LIN {X 0,Y 560.039,Z 923.26,A -85,B 0,C 180,E1 27100.284,E2 27100.284} C_VEL
LIN {X 0,Y 559.963,Z 930.88,A -85,B 0,C 180,E1 27098.213,E2 27098.213} C_VEL
LIN {X 0,Y 559.931,Z 936.64,A -85,B 0,C 180,E1 27096.151,E2 27096.151} C_VEL
LIN {X 0,Y 559.918,Z 940.7,A -85,B 0,C 180,E1 27094.096,E2 27094.096} C_VEL
LIN {X 0,Y 559.916,Z 943.21,A -85,B 0,C 180,E1 27091.944,E2 27091.944} C_VEL
LIN {X 0,Y 559.914,Z 943.994,A -85,B 0,C 180,E1 27089.898,E2 27089.898} C_VEL
LIN {X 0,Y 559.91,Z 943.066,A -85,B 0,C 180,E1 27087.748,E2 27087.748} C_VEL
LIN {X 0,Y 559.917,Z 940.522,A -85,B 0,C 180,E1 27085.699,E2 27085.699} C_VEL
LIN {X 0,Y 559.934,Z 936.354,A -85,B 0,C 180,E1 27083.644,E2 27083.644} C_VEL
LIN {X 0,Y 559.973,Z 930.444,A -85,B 0,C 180,E1 27081.57,E2 27081.57} C_VEL
LIN {X 0,Y 560.039,Z 923.202,A -85,B 0,C 180,E1 27079.612,E2 27079.612} C_VEL
LIN {X 0,Y 560.173,Z 913.998,A -85,B 0,C 180,E1 27077.632,E2 27077.632} C_VEL
LIN {X 0,Y 560.353,Z 903.373,A -85,B 0,C 180,E1 27075.745,E2 27075.745} C_VEL
LIN {X 0,Y 560.607,Z 891.369,A -85,B 0,C 180,E1 27073.952,E2 27073.952} C_VEL
LIN {X 0,Y 560.935,Z 877.981,A -85,B 0,C 180,E1 27072.253,E2 27072.253} C_VEL
LIN {X 0,Y 561.332,Z 863.174,A -85,B 0,C 180,E1 27070.652,E2 27070.652} C_VEL
LIN {X 0,Y 561.802,Z 846.535,A -85,B 0,C 180,E1 27069.126,E2 27069.126} C_VEL
LIN {X 0,Y 562.324,Z 828.625,A -85,B 0,C 180,E1 27067.745,E2 27067.745} C_VEL
LIN {X 0,Y 562.836,Z 809.963,A -85,B 0,C 180,E1 27066.551,E2 27066.551} C_VEL
LIN {X 0,Y 563.315,Z 791.261,A -85,B 0,C 180,E1 27065.571,E2 27065.571} C_VEL
LIN {X 0,Y 563.724,Z 772.173,A -85,B 0,C 180,E1 27064.766,E2 27064.766} C_VEL
LIN {X 0,Y 564.117,Z 751.599,A -85,B 0,C 180,E1 27064.104,E2 27064.104} C_VEL
LIN {X 0,Y 564.417,Z 731.328,A -85,B 0,C 180,E1 27063.645,E2 27063.645} C_VEL
LIN {X 0,Y 565.685,Z 480.008,A -85,B 0,C 180,E1 27060.141,E2 27060.141} C_VEL
LIN {X 0,Y 565.144,Z 474.616,A -85,B 0,C 180,E1 27060.032,E2 27060.032} C_VEL
LIN {X 0,Y 564.411,Z 469.546,A -85,B 0,C 180,E1 27059.882,E2 27059.882} C_VEL
LIN {X 0,Y 565.386,Z 421.661,A -85,B 0,C 180,E1 27056.633,E2 27056.633} C_VEL
LIN {X 0,Y 566.258,Z 392.209,A -85,B 0,C 180,E1 27054.54,E2 27054.54} C_VEL
LIN {X 0,Y 562.618,Z 383.241,A -85,B 0,C 180,E1 27053.53,E2 27053.53} C_VEL
LIN {X 0,Y 560.275,Z 377.562,A -85,B 0,C 180,E1 27052.843,E2 27052.843} C_VEL
LIN {X 0,Y 560.267,Z 377.245,A -85,B 0,C 180,E1 27051.868,E2 27051.868} C_VEL
LIN {X 0,Y 560.221,Z 377.251,A -85,B 0,C 180,E1 27048.808,E2 27048.808} C_VEL
LIN {X 0,Y 560.261,Z 377.247,A -85,B 0,C 180,E1 27045.549,E2 27045.549} C_VEL
LIN {X 0,Y 560.226,Z 377.259,A -85,B 0,C 180,E1 27042.426,E2 27042.426} C_VEL
LIN {X 0,Y 560.237,Z 377.262,A -85,B 0,C 180,E1 27039.051,E2 27039.051} C_VEL
LIN {X 0,Y 560.23,Z 377.247,A -85,B 0,C 180,E1 27036.051,E2 27036.051} C_VEL
LIN {X 0,Y 560.224,Z 377.259,A -85,B 0,C 180,E1 27032.605,E2 27032.605} C_VEL
LIN {X 0,Y 560.252,Z 377.242,A -85,B 0,C 180,E1 27029.51,E2 27029.51} C_VEL
LIN {X 0,Y 560.218,Z 377.258,A -85,B 0,C 180,E1 27026.272,E2 27026.272} C_VEL
LIN {X 0,Y 560.268,Z 377.258,A -85,B 0,C 180,E1 27023.118,E2 27023.118} C_VEL
LIN {X 0,Y 560.214,Z 377.26,A -85,B 0,C 180,E1 27019.932,E2 27019.932} C_VEL
LIN {X 0,Y 560.273,Z 377.257,A -85,B 0,C 180,E1 27016.805,E2 27016.805} C_VEL
LIN {X 0,Y 560.211,Z 377.26,A -85,B 0,C 180,E1 27013.627,E2 27013.627} C_VEL
LIN {X 0,Y 560.274,Z 377.254,A -85,B 0,C 180,E1 27010.48,E2 27010.48} C_VEL
LIN {X 0,Y 560.208,Z 377.257,A -85,B 0,C 180,E1 27007.28,E2 27007.28} C_VEL
LIN {X 0,Y 560.28,Z 377.258,A -85,B 0,C 180,E1 27004.094,E2 27004.094} C_VEL
LIN {X 0,Y 560.207,Z 377.259,A -85,B 0,C 180,E1 27000.921,E2 27000.921} C_VEL
LIN {X 0,Y 560.278,Z 377.261,A -85,B 0,C 180,E1 26997.75,E2 26997.75} C_VEL
LIN {X 0,Y 560.205,Z 377.26,A -85,B 0,C 180,E1 26994.572,E2 26994.572} C_VEL
LIN {X 0,Y 560.269,Z 377.26,A -85,B 0,C 180,E1 26991.37,E2 26991.37} C_VEL
LIN {X 0,Y 560.204,Z 377.253,A -85,B 0,C 180,E1 26988.261,E2 26988.261} C_VEL
LIN {X 0,Y 560.254,Z 377.258,A -85,B 0,C 180,E1 26985.003,E2 26985.003} C_VEL
LIN {X 0,Y 560.203,Z 377.256,A -85,B 0,C 180,E1 26982.015,E2 26982.015} C_VEL
LIN {X 0,Y 560.256,Z 377.257,A -85,B 0,C 180,E1 26978.76,E2 26978.76} C_VEL
LIN {X 0,Y 560.201,Z 377.256,A -85,B 0,C 180,E1 26975.764,E2 26975.764} C_VEL
LIN {X 0,Y 560.255,Z 377.262,A -85,B 0,C 180,E1 26972.496,E2 26972.496} C_VEL
LIN {X 0,Y 560.2,Z 377.25,A -85,B 0,C 180,E1 26969.425,E2 26969.425} C_VEL
LIN {X 0,Y 560.245,Z 377.256,A -85,B 0,C 180,E1 26966.164,E2 26966.164} C_VEL
LIN {X 0,Y 560.202,Z 377.263,A -85,B 0,C 180,E1 26963.092,E2 26963.092} C_VEL
LIN {X 0,Y 560.233,Z 377.255,A -85,B 0,C 180,E1 26959.806,E2 26959.806} C_VEL
LIN {X 0,Y 560.196,Z 377.245,A -85,B 0,C 180,E1 26956.876,E2 26956.876} C_VEL
LIN {X 0,Y 560.287,Z 377.452,A -85,B 0,C 180,E1 26956.18,E2 26956.18} C_VEL
LIN {X 0,Y 561.118,Z 379.974,A -85,B 0,C 180,E1 26955.899,E2 26955.899} C_VEL
LIN {X 0,Y 564.918,Z 386.463,A -85,B 0,C 180,E1 26955.214,E2 26955.214} C_VEL
LIN {X 0,Y 570.593,Z 397.019,A -85,B 0,C 180,E1 26954.056,E2 26954.056} C_VEL
LIN {X 0,Y 569.301,Z 451.788,A -85,B 0,C 180,E1 26951.15,E2 26951.15} C_VEL
LIN {X 0,Y 569.17,Z 466.355,A -85,B 0,C 180,E1 26950.418,E2 26950.418} C_VEL
LIN {X 0,Y 570.273,Z 475.671,A -85,B 0,C 180,E1 26950.173,E2 26950.173} C_VEL
LIN {X 0,Y 568.787,Z 680.489,A -85,B 0,C 180,E1 26947.054,E2 26947.054} C_VEL
LIN {X 0,Y 567.809,Z 815.971,A -85,B 0,C 180,E1 26945.018,E2 26945.018} C_VEL
LIN {X 0,Y 567.322,Z 839.745,A -85,B 0,C 180,E1 26944.473,E2 26944.473} C_VEL
LIN {X 0,Y 566.852,Z 861.613,A -85,B 0,C 180,E1 26943.785,E2 26943.785} C_VEL
LIN {X 0,Y 566.166,Z 883.682,A -85,B 0,C 180,E1 26942.892,E2 26942.892} C_VEL
LIN {X 0,Y 565.506,Z 904.783,A -85,B 0,C 180,E1 26941.855,E2 26941.855} C_VEL
LIN {X 0,Y 564.723,Z 925.843,A -85,B 0,C 180,E1 26940.605,E2 26940.605} C_VEL
LIN {X 0,Y 563.96,Z 946.403,A -85,B 0,C 180,E1 26939.18,E2 26939.18} C_VEL
LIN {X 0,Y 563.25,Z 964.586,A -85,B 0,C 180,E1 26937.716,E2 26937.716} C_VEL
LIN {X 0,Y 562.525,Z 983.959,A -85,B 0,C 180,E1 26935.923,E2 26935.923} C_VEL
LIN {X 0,Y 561.904,Z 1001.171,A -85,B 0,C 180,E1 26934.101,E2 26934.101} C_VEL
LIN {X 0,Y 561.359,Z 1017.098,A -85,B 0,C 180,E1 26932.152,E2 26932.152} C_VEL
LIN {X 0,Y 560.903,Z 1032.335,A -85,B 0,C 180,E1 26930.015,E2 26930.015} C_VEL
LIN {X 0,Y 560.562,Z 1045.006,A -85,B 0,C 180,E1 26927.974,E2 26927.974} C_VEL
LIN {X 0,Y 560.296,Z 1056.318,A -85,B 0,C 180,E1 26925.845,E2 26925.845} C_VEL
LIN {X 0,Y 560.126,Z 1065.995,A -85,B 0,C 180,E1 26923.734,E2 26923.734} C_VEL
LIN {X 0,Y 560.023,Z 1074.34,A -85,B 0,C 180,E1 26921.535,E2 26921.535} C_VEL
LIN {X 0,Y 559.945,Z 1080.869,A -85,B 0,C 180,E1 26919.455,E2 26919.455} C_VEL
LIN {X 0,Y 559.899,Z 1086.634,A -85,B 0,C 180,E1 26917.078,E2 26917.078} C_VEL
LIN {X 0,Y 559.911,Z 1090.276,A -85,B 0,C 180,E1 26915.02,E2 26915.02} C_VEL
LIN {X 0,Y 559.913,Z 1092.988,A -85,B 0,C 180,E1 26912.559,E2 26912.559} C_VEL
LIN {X 0,Y 559.887,Z 1093.917,A -85,B 0,C 180,E1 26910.409,E2 26910.409} C_VEL
LIN {X 0,Y 559.912,Z 1093.324,A -85,B 0,C 180,E1 26907.953,E2 26907.953} C_VEL
LIN {X 0,Y 559.912,Z 1091.276,A -85,B 0,C 180,E1 26905.699,E2 26905.699} C_VEL
LIN {X 0,Y 559.914,Z 1087.46,A -85,B 0,C 180,E1 26903.334,E2 26903.334} C_VEL
LIN {X 0,Y 559.949,Z 1082.806,A -85,B 0,C 180,E1 26901.27,E2 26901.27} C_VEL
LIN {X 0,Y 559.994,Z 1075.764,A -85,B 0,C 180,E1 26898.882,E2 26898.882} C_VEL
LIN {X 0,Y 560.096,Z 1068.109,A -85,B 0,C 180,E1 26896.791,E2 26896.791} C_VEL
LIN {X 0,Y 560.276,Z 1057.882,A -85,B 0,C 180,E1 26894.473,E2 26894.473} C_VEL
LIN {X 0,Y 560.533,Z 1046.819,A -85,B 0,C 180,E1 26892.348,E2 26892.348} C_VEL
LIN {X 0,Y 560.861,Z 1033.752,A -85,B 0,C 180,E1 26890.201,E2 26890.201} C_VEL
LIN {X 0,Y 561.294,Z 1019.336,A -85,B 0,C 180,E1 26888.136,E2 26888.136} C_VEL
LIN {X 0,Y 561.8,Z 1003.941,A -85,B 0,C 180,E1 26886.227,E2 26886.227} C_VEL
LIN {X 0,Y 562.437,Z 986.114,A -85,B 0,C 180,E1 26884.293,E2 26884.293} C_VEL
LIN {X 0,Y 563.119,Z 968.256,A -85,B 0,C 180,E1 26882.595,E2 26882.595} C_VEL
LIN {X 0,Y 563.847,Z 949.336,A -85,B 0,C 180,E1 26881.046,E2 26881.046} C_VEL
LIN {X 0,Y 564.609,Z 928.601,A -85,B 0,C 180,E1 26879.57,E2 26879.57} C_VEL
LIN {X 0,Y 565.354,Z 908.827,A -85,B 0,C 180,E1 26878.373,E2 26878.373} C_VEL
LIN {X 0,Y 566.073,Z 886.169,A -85,B 0,C 180,E1 26877.22,E2 26877.22} C_VEL
LIN {X 0,Y 566.734,Z 865.501,A -85,B 0,C 180,E1 26876.36,E2 26876.36} C_VEL
LIN {X 0,Y 567.276,Z 842.338,A -85,B 0,C 180,E1 26875.6,E2 26875.6} C_VEL
LIN {X 0,Y 567.747,Z 820.122,A -85,B 0,C 180,E1 26875.058,E2 26875.058} C_VEL
LIN {X 0,Y 568.087,Z 782.758,A -85,B 0,C 180,E1 26874.465,E2 26874.465} C_VEL
LIN {X 0,Y 569.521,Z 575.861,A -85,B 0,C 180,E1 26871.366,E2 26871.366} C_VEL
LIN {X 0,Y 570.109,Z 472.892,A -85,B 0,C 180,E1 26869.768,E2 26869.768} C_VEL
LIN {X 0,Y 569.041,Z 464.13,A -85,B 0,C 180,E1 26869.491,E2 26869.491} C_VEL
LIN {X 0,Y 570.379,Z 406.466,A -85,B 0,C 180,E1 26866.455,E2 26866.455} C_VEL
LIN {X 0,Y 570.536,Z 396.902,A -85,B 0,C 180,E1 26865.932,E2 26865.932} C_VEL
LIN {X 0,Y 564.905,Z 386.448,A -85,B 0,C 180,E1 26864.784,E2 26864.784} C_VEL
LIN {X 0,Y 562.383,Z 381.983,A -85,B 0,C 180,E1 26864.323,E2 26864.323} C_VEL
LIN {X 0,Y 560.392,Z 377.966,A -85,B 0,C 180,E1 26863.909,E2 26863.909} C_VEL
LIN {X 0,Y 560.241,Z 377.261,A -85,B 0,C 180,E1 26863.683,E2 26863.683} C_VEL
LIN {X 0,Y 560.2,Z 377.267,A -85,B 0,C 180,E1 26860.651,E2 26860.651} C_VEL
LIN {X 0,Y 560.236,Z 377.263,A -85,B 0,C 180,E1 26857.358,E2 26857.358} C_VEL
LIN {X 0,Y 560.201,Z 377.256,A -85,B 0,C 180,E1 26854.333,E2 26854.333} C_VEL
LIN {X 0,Y 560.231,Z 377.248,A -85,B 0,C 180,E1 26851.049,E2 26851.049} C_VEL
LIN {X 0,Y 560.203,Z 377.263,A -85,B 0,C 180,E1 26848.111,E2 26848.111} C_VEL
LIN {X 0,Y 560.236,Z 377.255,A -85,B 0,C 180,E1 26844.797,E2 26844.797} C_VEL
LIN {X 0,Y 560.202,Z 377.262,A -85,B 0,C 180,E1 26841.857,E2 26841.857} C_VEL
LIN {X 0,Y 560.248,Z 377.254,A -85,B 0,C 180,E1 26838.618,E2 26838.618} C_VEL
LIN {X 0,Y 560.202,Z 377.261,A -85,B 0,C 180,E1 26835.635,E2 26835.635} C_VEL
LIN {X 0,Y 560.266,Z 377.245,A -85,B 0,C 180,E1 26832.47,E2 26832.47} C_VEL
LIN {X 0,Y 560.204,Z 377.26,A -85,B 0,C 180,E1 26829.347,E2 26829.347} C_VEL
LIN {X 0,Y 560.261,Z 377.258,A -85,B 0,C 180,E1 26826.147,E2 26826.147} C_VEL
LIN {X 0,Y 560.204,Z 377.259,A -85,B 0,C 180,E1 26823.069,E2 26823.069} C_VEL
LIN {X 0,Y 560.252,Z 377.259,A -85,B 0,C 180,E1 26819.795,E2 26819.795} C_VEL
LIN {X 0,Y 560.207,Z 377.259,A -85,B 0,C 180,E1 26816.726,E2 26816.726} C_VEL
LIN {X 0,Y 560.242,Z 377.255,A -85,B 0,C 180,E1 26813.441,E2 26813.441} C_VEL
LIN {X 0,Y 560.21,Z 377.261,A -85,B 0,C 180,E1 26810.445,E2 26810.445} C_VEL
LIN {X 0,Y 560.238,Z 377.259,A -85,B 0,C 180,E1 26807.109,E2 26807.109} C_VEL
LIN {X 0,Y 560.21,Z 377.259,A -85,B 0,C 180,E1 26804.152,E2 26804.152} C_VEL
LIN {X 0,Y 560.238,Z 377.258,A -85,B 0,C 180,E1 26800.829,E2 26800.829} C_VEL
LIN {X 0,Y 560.213,Z 377.258,A -85,B 0,C 180,E1 26797.867,E2 26797.867} C_VEL
LIN {X 0,Y 560.219,Z 377.26,A -85,B 0,C 180,E1 26796.413,E2 26796.413} C_VEL
LIN {X 0,Y 559.219,Z 377.387,A -85,B 0,C 180,E1 26795.625,E2 26795.625} C_VEL
LIN {X 0,Y 552.8,Z 378.196,A -85,B 0,C 180,E1 26793.356,E2 26793.356} C_VEL
LIN {X 0,Y 552.341,Z 378.247,A -85,B 0,C 180,E1 26792.837,E2 26792.837} C_VEL
LIN {X 0,Y 552.269,Z 378.232,A -85,B 0,C 180,E1 26789.661,E2 26789.661} C_VEL
LIN {X 0,Y 552.323,Z 378.245,A -85,B 0,C 180,E1 26786.381,E2 26786.381} C_VEL
LIN {X 0,Y 552.273,Z 378.237,A -85,B 0,C 180,E1 26783.312,E2 26783.312} C_VEL
LIN {X 0,Y 552.312,Z 378.237,A -85,B 0,C 180,E1 26780.009,E2 26780.009} C_VEL
LIN {X 0,Y 552.278,Z 378.251,A -85,B 0,C 180,E1 26776.958,E2 26776.958} C_VEL
LIN {X 0,Y 552.299,Z 378.244,A -85,B 0,C 180,E1 26773.602,E2 26773.602} C_VEL
LIN {X 0,Y 552.288,Z 378.235,A -85,B 0,C 180,E1 26770.503,E2 26770.503} C_VEL
LIN {X 0,Y 552.376,Z 378.457,A -85,B 0,C 180,E1 26767.751,E2 26767.751} C_VEL
LIN {X 0,Y 553.454,Z 381.481,A -85,B 0,C 180,E1 26767.354,E2 26767.354} C_VEL
LIN {X 0,Y 558.546,Z 392.913,A -85,B 0,C 180,E1 26765.989,E2 26765.989} C_VEL
LIN {X 0,Y 559.571,Z 396.38,A -85,B 0,C 180,E1 26765.627,E2 26765.627} C_VEL
LIN {X 0,Y 557.981,Z 436.754,A -85,B 0,C 180,E1 26762.702,E2 26762.702} C_VEL
LIN {X 0,Y 557.331,Z 470.637,A -85,B 0,C 180,E1 26760.404,E2 26760.404} C_VEL
LIN {X 0,Y 558.746,Z 480.648,A -85,B 0,C 180,E1 26760.168,E2 26760.168} C_VEL
LIN {X 0,Y 557.241,Z 731.515,A -85,B 0,C 180,E1 26756.627,E2 26756.627} C_VEL
LIN {X 0,Y 556.888,Z 751.851,A -85,B 0,C 180,E1 26756.16,E2 26756.16} C_VEL
LIN {X 0,Y 556.453,Z 771.613,A -85,B 0,C 180,E1 26755.518,E2 26755.518} C_VEL
LIN {X 0,Y 555.939,Z 791.709,A -85,B 0,C 180,E1 26754.662,E2 26754.662} C_VEL
LIN {X 0,Y 555.372,Z 810.318,A -85,B 0,C 180,E1 26753.671,E2 26753.671} C_VEL
LIN {X 0,Y 554.773,Z 828.915,A -85,B 0,C 180,E1 26752.463,E2 26752.463} C_VEL
LIN {X 0,Y 554.194,Z 845.971,A -85,B 0,C 180,E1 26751.131,E2 26751.131} C_VEL
LIN {X 0,Y 553.646,Z 862.259,A -85,B 0,C 180,E1 26749.628,E2 26749.628} C_VEL
LIN {X 0,Y 553.164,Z 877.209,A -85,B 0,C 180,E1 26748.004,E2 26748.004} C_VEL
LIN {X 0,Y 552.772,Z 890.722,A -85,B 0,C 180,E1 26746.282,E2 26746.282} C_VEL
LIN {X 0,Y 552.439,Z 903.473,A -85,B 0,C 180,E1 26744.357,E2 26744.357} C_VEL
LIN {X 0,Y 552.223,Z 914.076,A -85,B 0,C 180,E1 26742.443,E2 26742.443} C_VEL
LIN {X 0,Y 552.07,Z 923.263,A -85,B 0,C 180,E1 26740.435,E2 26740.435} C_VEL
LIN {X 0,Y 551.978,Z 930.882,A -85,B 0,C 180,E1 26738.332,E2 26738.332} C_VEL
LIN {X 0,Y 551.937,Z 936.642,A -85,B 0,C 180,E1 26736.24,E2 26736.24} C_VEL
LIN {X 0,Y 551.919,Z 940.702,A -85,B 0,C 180,E1 26734.156,E2 26734.156} C_VEL
LIN {X 0,Y 551.916,Z 943.21,A -85,B 0,C 180,E1 26731.973,E2 26731.973} C_VEL
LIN {X 0,Y 551.914,Z 943.994,A -85,B 0,C 180,E1 26729.896,E2 26729.896} C_VEL
LIN {X 0,Y 551.909,Z 943.065,A -85,B 0,C 180,E1 26727.716,E2 26727.716} C_VEL
LIN {X 0,Y 551.917,Z 940.52,A -85,B 0,C 180,E1 26725.636,E2 26725.636} C_VEL
LIN {X 0,Y 551.938,Z 936.353,A -85,B 0,C 180,E1 26723.551,E2 26723.551} C_VEL
LIN {X 0,Y 551.985,Z 930.478,A -85,B 0,C 180,E1 26721.458,E2 26721.458} C_VEL
LIN {X 0,Y 552.071,Z 923.2,A -85,B 0,C 180,E1 26719.46,E2 26719.46} C_VEL
LIN {X 0,Y 552.232,Z 913.73,A -85,B 0,C 180,E1 26717.397,E2 26717.397} C_VEL
LIN {X 0,Y 552.444,Z 903.349,A -85,B 0,C 180,E1 26715.533,E2 26715.533} C_VEL
LIN {X 0,Y 552.751,Z 891.363,A -85,B 0,C 180,E1 26713.717,E2 26713.717} C_VEL
LIN {X 0,Y 553.154,Z 877.577,A -85,B 0,C 180,E1 26711.949,E2 26711.949} C_VEL
LIN {X 0,Y 553.635,Z 862.616,A -85,B 0,C 180,E1 26710.317,E2 26710.317} C_VEL
LIN {X 0,Y 554.165,Z 846.804,A -85,B 0,C 180,E1 26708.847,E2 26708.847} C_VEL
LIN {X 0,Y 554.755,Z 829.363,A -85,B 0,C 180,E1 26707.48,E2 26707.48} C_VEL
LIN {X 0,Y 555.326,Z 811.752,A -85,B 0,C 180,E1 26706.327,E2 26706.327} C_VEL
LIN {X 0,Y 555.904,Z 792.802,A -85,B 0,C 180,E1 26705.301,E2 26705.301} C_VEL
LIN {X 0,Y 556.425,Z 772.659,A -85,B 0,C 180,E1 26704.431,E2 26704.431} C_VEL
LIN {X 0,Y 556.881,Z 752.484,A -85,B 0,C 180,E1 26703.767,E2 26703.767} C_VEL
LIN {X 0,Y 557.238,Z 732.116,A -85,B 0,C 180,E1 26703.293,E2 26703.293} C_VEL
LIN {X 0,Y 558.712,Z 485.739,A -85,B 0,C 180,E1 26699.814,E2 26699.814} C_VEL
LIN {X 0,Y 558.499,Z 477.663,A -85,B 0,C 180,E1 26699.684,E2 26699.684} C_VEL
LIN {X 0,Y 557.255,Z 469.588,A -85,B 0,C 180,E1 26699.457,E2 26699.457} C_VEL
LIN {X 0,Y 558.441,Z 423.706,A -85,B 0,C 180,E1 26696.286,E2 26696.286} C_VEL
LIN {X 0,Y 559.556,Z 395.575,A -85,B 0,C 180,E1 26694.218,E2 26694.218} C_VEL
LIN {X 0,Y 555.395,Z 385.624,A -85,B 0,C 180,E1 26693.065,E2 26693.065} C_VEL
LIN {X 0,Y 552.391,Z 378.546,A -85,B 0,C 180,E1 26692.185,E2 26692.185} C_VEL
LIN {X 0,Y 552.284,Z 378.249,A -85,B 0,C 180,E1 26691.287,E2 26691.287} C_VEL
LIN {X 0,Y 552.34,Z 378.238,A -85,B 0,C 180,E1 26688.074,E2 26688.074} C_VEL
LIN {X 0,Y 552.281,Z 378.243,A -85,B 0,C 180,E1 26684.79,E2 26684.79} C_VEL
LIN {X 0,Y 552.333,Z 378.233,A -85,B 0,C 180,E1 26681.495,E2 26681.495} C_VEL
LIN {X 0,Y 552.281,Z 378.25,A -85,B 0,C 180,E1 26678.379,E2 26678.379} C_VEL
LIN {X 0,Y 552.311,Z 378.24,A -85,B 0,C 180,E1 26675.021,E2 26675.021} C_VEL
LIN {X 0,Y 552.291,Z 378.246,A -85,B 0,C 180,E1 26671.889,E2 26671.889} C_VEL
LIN {X 0,Y 552.284,Z 378.248,A -85,B 0,C 180,E1 26668.434,E2 26668.434} C_VEL
LIN {X 0,Y 552.308,Z 378.245,A -85,B 0,C 180,E1 26665.397,E2 26665.397} C_VEL
LIN {X 0,Y 552.277,Z 378.246,A -85,B 0,C 180,E1 26662.036,E2 26662.036} C_VEL
LIN {X 0,Y 552.331,Z 378.246,A -85,B 0,C 180,E1 26658.907,E2 26658.907} C_VEL
LIN {X 0,Y 552.272,Z 378.247,A -85,B 0,C 180,E1 26655.65,E2 26655.65} C_VEL
LIN {X 0,Y 552.345,Z 378.248,A -85,B 0,C 180,E1 26652.44,E2 26652.44} C_VEL
LIN {X 0,Y 552.271,Z 378.249,A -85,B 0,C 180,E1 26649.273,E2 26649.273} C_VEL
LIN {X 0,Y 552.335,Z 378.249,A -85,B 0,C 180,E1 26646.027,E2 26646.027} C_VEL
LIN {X 0,Y 552.27,Z 378.246,A -85,B 0,C 180,E1 26642.906,E2 26642.906} C_VEL
LIN {X 0,Y 552.326,Z 378.246,A -85,B 0,C 180,E1 26639.689,E2 26639.689} C_VEL
LIN {X 0,Y 552.27,Z 378.247,A -85,B 0,C 180,E1 26636.575,E2 26636.575} C_VEL
LIN {X 0,Y 552.303,Z 378.247,A -85,B 0,C 180,E1 26633.243,E2 26633.243} C_VEL
LIN {X 0,Y 552.272,Z 378.249,A -85,B 0,C 180,E1 26630.202,E2 26630.202} C_VEL
LIN {X 0,Y 552.285,Z 378.234,A -85,B 0,C 180,E1 26626.814,E2 26626.814} C_VEL
LIN {X 0,Y 552.272,Z 378.249,A -85,B 0,C 180,E1 26623.919,E2 26623.919} C_VEL
LIN {X 0,Y 552.282,Z 378.233,A -85,B 0,C 180,E1 26620.542,E2 26620.542} C_VEL
LIN {X 0,Y 552.269,Z 378.25,A -85,B 0,C 180,E1 26617.655,E2 26617.655} C_VEL
LIN {X 0,Y 552.28,Z 378.238,A -85,B 0,C 180,E1 26614.247,E2 26614.247} C_VEL
LIN {X 0,Y 552.272,Z 378.251,A -85,B 0,C 180,E1 26611.33,E2 26611.33} C_VEL
LIN {X 0,Y 552.27,Z 378.252,A -85,B 0,C 180,E1 26607.841,E2 26607.841} C_VEL
LIN {X 0,Y 552.284,Z 378.238,A -85,B 0,C 180,E1 26604.851,E2 26604.851} C_VEL
LIN {X 0,Y 552.27,Z 378.244,A -85,B 0,C 180,E1 26601.612,E2 26601.612} C_VEL
LIN {X 0,Y 552.28,Z 378.254,A -85,B 0,C 180,E1 26598.639,E2 26598.639} C_VEL
LIN {X 0,Y 552.294,Z 378.486,A -85,B 0,C 180,E1 26596.847,E2 26596.847} C_VEL
LIN {X 0,Y 553.472,Z 381.544,A -85,B 0,C 180,E1 26596.506,E2 26596.506} C_VEL
LIN {X 0,Y 554.698,Z 383.43,A -85,B 0,C 180,E1 26596.288,E2 26596.288} C_VEL
LIN {X 0,Y 558.901,Z 391.38,A -85,B 0,C 180,E1 26595.471,E2 26595.471} C_VEL
LIN {X 0,Y 564.408,Z 400.854,A -85,B 0,C 180,E1 26594.446,E2 26594.446} C_VEL
LIN {X 0,Y 563.029,Z 452.214,A -85,B 0,C 180,E1 26591.687,E2 26591.687} C_VEL
LIN {X 0,Y 562.845,Z 466.387,A -85,B 0,C 180,E1 26590.968,E2 26590.968} C_VEL
LIN {X 0,Y 564.146,Z 477.002,A -85,B 0,C 180,E1 26590.678,E2 26590.678} C_VEL
LIN {X 0,Y 562.392,Z 681.557,A -85,B 0,C 180,E1 26587.531,E2 26587.531} C_VEL
LIN {X 0,Y 561.248,Z 816.077,A -85,B 0,C 180,E1 26585.487,E2 26585.487} C_VEL
LIN {X 0,Y 560.693,Z 839.743,A -85,B 0,C 180,E1 26584.939,E2 26584.939} C_VEL
LIN {X 0,Y 560.123,Z 861.657,A -85,B 0,C 180,E1 26584.245,E2 26584.245} C_VEL
LIN {X 0,Y 559.344,Z 883.679,A -85,B 0,C 180,E1 26583.345,E2 26583.345} C_VEL
LIN {X 0,Y 558.545,Z 904.783,A -85,B 0,C 180,E1 26582.3,E2 26582.3} C_VEL
LIN {X 0,Y 557.68,Z 925.046,A -85,B 0,C 180,E1 26581.088,E2 26581.088} C_VEL
LIN {X 0,Y 556.794,Z 944.93,A -85,B 0,C 180,E1 26579.711,E2 26579.711} C_VEL
LIN {X 0,Y 555.952,Z 963.507,A -85,B 0,C 180,E1 26578.208,E2 26578.208} C_VEL
LIN {X 0,Y 555.084,Z 982.792,A -85,B 0,C 180,E1 26576.418,E2 26576.418} C_VEL
LIN {X 0,Y 554.356,Z 999.661,A -85,B 0,C 180,E1 26574.623,E2 26574.623} C_VEL
LIN {X 0,Y 553.688,Z 1015.994,A -85,B 0,C 180,E1 26572.621,E2 26572.621} C_VEL
LIN {X 0,Y 553.14,Z 1030.919,A -85,B 0,C 180,E1 26570.529,E2 26570.529} C_VEL
LIN {X 0,Y 552.723,Z 1043.734,A -85,B 0,C 180,E1 26568.456,E2 26568.456} C_VEL
LIN {X 0,Y 552.396,Z 1055.798,A -85,B 0,C 180,E1 26566.186,E2 26566.186} C_VEL
LIN {X 0,Y 552.204,Z 1065.076,A -85,B 0,C 180,E1 26564.149,E2 26564.149} C_VEL
LIN {X 0,Y 552.057,Z 1073.985,A -85,B 0,C 180,E1 26561.81,E2 26561.81} C_VEL
LIN {X 0,Y 551.951,Z 1080.565,A -85,B 0,C 180,E1 26559.699,E2 26559.699} C_VEL
LIN {X 0,Y 551.906,Z 1086.427,A -85,B 0,C 180,E1 26557.286,E2 26557.286} C_VEL
LIN {X 0,Y 551.913,Z 1090.117,A -85,B 0,C 180,E1 26555.197,E2 26555.197} C_VEL
LIN {X 0,Y 551.897,Z 1092.852,A -85,B 0,C 180,E1 26552.804,E2 26552.804} C_VEL
LIN {X 0,Y 551.883,Z 1093.85,A -85,B 0,C 180,E1 26550.727,E2 26550.727} C_VEL
LIN {X 0,Y 551.906,Z 1093.657,A -85,B 0,C 180,E1 26548.443,E2 26548.443} C_VEL
LIN {X 0,Y 551.915,Z 1091.729,A -85,B 0,C 180,E1 26546.053,E2 26546.053} C_VEL
LIN {X 0,Y 551.93,Z 1088.287,A -85,B 0,C 180,E1 26543.655,E2 26543.655} C_VEL
LIN {X 0,Y 551.952,Z 1083.571,A -85,B 0,C 180,E1 26541.457,E2 26541.457} C_VEL
LIN {X 0,Y 552.011,Z 1077.178,A -85,B 0,C 180,E1 26539.142,E2 26539.142} C_VEL
LIN {X 0,Y 552.125,Z 1069.337,A -85,B 0,C 180,E1 26536.917,E2 26536.917} C_VEL
LIN {X 0,Y 552.325,Z 1059.944,A -85,B 0,C 180,E1 26534.674,E2 26534.674} C_VEL
LIN {X 0,Y 552.597,Z 1048.848,A -85,B 0,C 180,E1 26532.465,E2 26532.465} C_VEL
LIN {X 0,Y 552.987,Z 1035.867,A -85,B 0,C 180,E1 26530.238,E2 26530.238} C_VEL
LIN {X 0,Y 553.48,Z 1021.778,A -85,B 0,C 180,E1 26528.152,E2 26528.152} C_VEL
LIN {X 0,Y 554.1,Z 1005.801,A -85,B 0,C 180,E1 26526.102,E2 26526.102} C_VEL
LIN {X 0,Y 554.813,Z 989.039,A -85,B 0,C 180,E1 26524.217,E2 26524.217} C_VEL
LIN {X 0,Y 555.57,Z 971.797,A -85,B 0,C 180,E1 26522.529,E2 26522.529} C_VEL
LIN {X 0,Y 556.486,Z 951.899,A -85,B 0,C 180,E1 26520.833,E2 26520.833} C_VEL
LIN {X 0,Y 557.323,Z 933.12,A -85,B 0,C 180,E1 26519.444,E2 26519.444} C_VEL
LIN {X 0,Y 558.201,Z 912.828,A -85,B 0,C 180,E1 26518.162,E2 26518.162} C_VEL
LIN {X 0,Y 559.039,Z 892.43,A -85,B 0,C 180,E1 26517.063,E2 26517.063} C_VEL
LIN {X 0,Y 559.785,Z 870.673,A -85,B 0,C 180,E1 26516.101,E2 26516.101} C_VEL
LIN {X 0,Y 560.536,Z 848.173,A -85,B 0,C 180,E1 26515.302,E2 26515.302} C_VEL
LIN {X 0,Y 561.01,Z 825.427,A -85,B 0,C 180,E1 26514.704,E2 26514.704} C_VEL
LIN {X 0,Y 561.448,Z 799.681,A -85,B 0,C 180,E1 26514.241,E2 26514.241} C_VEL
LIN {X 0,Y 563.188,Z 586.683,A -85,B 0,C 180,E1 26511.023,E2 26511.023} C_VEL
LIN {X 0,Y 563.993,Z 474.426,A -85,B 0,C 180,E1 26509.266,E2 26509.266} C_VEL
LIN {X 0,Y 562.722,Z 464.635,A -85,B 0,C 180,E1 26508.963,E2 26508.963} C_VEL
LIN {X 0,Y 564.274,Z 407.703,A -85,B 0,C 180,E1 26505.934,E2 26505.934} C_VEL
LIN {X 0,Y 564.408,Z 400.854,A -85,B 0,C 180,E1 26505.554,E2 26505.554} C_VEL
LIN {X 0,Y 558.903,Z 391.381,A -85,B 0,C 180,E1 26504.529,E2 26504.529} C_VEL
LIN {X 0,Y 554.006,Z 382.276,A -85,B 0,C 180,E1 26503.584,E2 26503.584} C_VEL
LIN {X 0,Y 552.343,Z 378.76,A -85,B 0,C 180,E1 26503.2,E2 26503.2} C_VEL
LIN {X 0,Y 552.255,Z 378.231,A -85,B 0,C 180,E1 26502.902,E2 26502.902} C_VEL
LIN {X 0,Y 552.329,Z 378.231,A -85,B 0,C 180,E1 26499.703,E2 26499.703} C_VEL
LIN {X 0,Y 552.258,Z 378.253,A -85,B 0,C 180,E1 26496.559,E2 26496.559} C_VEL
LIN {X 0,Y 552.325,Z 378.251,A -85,B 0,C 180,E1 26493.389,E2 26493.389} C_VEL
LIN {X 0,Y 552.261,Z 378.238,A -85,B 0,C 180,E1 26490.219,E2 26490.219} C_VEL
LIN {X 0,Y 552.313,Z 378.241,A -85,B 0,C 180,E1 26487.025,E2 26487.025} C_VEL
LIN {X 0,Y 552.265,Z 378.246,A -85,B 0,C 180,E1 26483.894,E2 26483.894} C_VEL
LIN {X 0,Y 552.291,Z 378.235,A -85,B 0,C 180,E1 26480.561,E2 26480.561} C_VEL
LIN {X 0,Y 552.267,Z 378.246,A -85,B 0,C 180,E1 26477.598,E2 26477.598} C_VEL
LIN {X 0,Y 552.29,Z 378.236,A -85,B 0,C 180,E1 26474.253,E2 26474.253} C_VEL
LIN {X 0,Y 552.27,Z 378.241,A -85,B 0,C 180,E1 26471.275,E2 26471.275} C_VEL
LIN {X 0,Y 552.283,Z 378.244,A -85,B 0,C 180,E1 26467.908,E2 26467.908} C_VEL
LIN {X 0,Y 552.272,Z 378.249,A -85,B 0,C 180,E1 26464.985,E2 26464.985} C_VEL
LIN {X 0,Y 552.28,Z 378.247,A -85,B 0,C 180,E1 26461.556,E2 26461.556} C_VEL
LIN {X 0,Y 552.277,Z 378.25,A -85,B 0,C 180,E1 26458.651,E2 26458.651} C_VEL
LIN {X 0,Y 552.276,Z 378.249,A -85,B 0,C 180,E1 26455.223,E2 26455.223} C_VEL
LIN {X 0,Y 552.284,Z 378.246,A -85,B 0,C 180,E1 26452.301,E2 26452.301} C_VEL
LIN {X 0,Y 552.274,Z 378.244,A -85,B 0,C 180,E1 26448.892,E2 26448.892} C_VEL
LIN {X 0,Y 552.301,Z 378.251,A -85,B 0,C 180,E1 26445.853,E2 26445.853} C_VEL
LIN {X 0,Y 552.272,Z 378.248,A -85,B 0,C 180,E1 26442.51,E2 26442.51} C_VEL
LIN {X 0,Y 552.333,Z 378.25,A -85,B 0,C 180,E1 26439.329,E2 26439.329} C_VEL
LIN {X 0,Y 552.268,Z 378.25,A -85,B 0,C 180,E1 26436.075,E2 26436.075} C_VEL
LIN {X 0,Y 552.341,Z 378.247,A -85,B 0,C 180,E1 26432.837,E2 26432.837} C_VEL
LIN {X 0,Y 551.295,Z 378.37,A -85,B 0,C 180,E1 26432.038,E2 26432.038} C_VEL
LIN {X 0,Y 544.842,Z 379.156,A -85,B 0,C 180,E1 26429.795,E2 26429.795} C_VEL
LIN {X 0,Y 544.356,Z 379.218,A -85,B 0,C 180,E1 26429.211,E2 26429.211} C_VEL
LIN {X 0,Y 544.337,Z 379.235,A -85,B 0,C 180,E1 26425.8,E2 26425.8} C_VEL
LIN {X 0,Y 544.399,Z 379.227,A -85,B 0,C 180,E1 26422.56,E2 26422.56} C_VEL
LIN {X 0,Y 544.333,Z 379.226,A -85,B 0,C 180,E1 26419.301,E2 26419.301} C_VEL
LIN {X 0,Y 544.396,Z 379.23,A -85,B 0,C 180,E1 26416.032,E2 26416.032} C_VEL
LIN {X 0,Y 544.338,Z 379.241,A -85,B 0,C 180,E1 26412.815,E2 26412.815} C_VEL
LIN {X 0,Y 544.365,Z 379.233,A -85,B 0,C 180,E1 26409.459,E2 26409.459} C_VEL
LIN {X 0,Y 544.39,Z 379.519,A -85,B 0,C 180,E1 26408.425,E2 26408.425} C_VEL
LIN {X 0,Y 545.658,Z 382.645,A -85,B 0,C 180,E1 26408.002,E2 26408.002} C_VEL
LIN {X 0,Y 552.336,Z 397.695,A -85,B 0,C 180,E1 26406.167,E2 26406.167} C_VEL
LIN {X 0,Y 552.916,Z 400.106,A -85,B 0,C 180,E1 26405.925,E2 26405.925} C_VEL
LIN {X 0,Y 550.902,Z 444.856,A -85,B 0,C 180,E1 26402.633,E2 26402.633} C_VEL
LIN {X 0,Y 550.157,Z 470.371,A -85,B 0,C 180,E1 26400.851,E2 26400.851} C_VEL
LIN {X 0,Y 551.825,Z 481.83,A -85,B 0,C 180,E1 26400.57,E2 26400.57} C_VEL
LIN {X 0,Y 550.09,Z 731.343,A -85,B 0,C 180,E1 26397.005,E2 26397.005} C_VEL
LIN {X 0,Y 549.685,Z 751.726,A -85,B 0,C 180,E1 26396.534,E2 26396.534} C_VEL
LIN {X 0,Y 549.193,Z 771.63,A -85,B 0,C 180,E1 26395.88,E2 26395.88} C_VEL
LIN {X 0,Y 548.594,Z 791.721,A -85,B 0,C 180,E1 26395.014,E2 26395.014} C_VEL
LIN {X 0,Y 547.937,Z 810.327,A -85,B 0,C 180,E1 26394.012,E2 26394.012} C_VEL
LIN {X 0,Y 547.253,Z 828.924,A -85,B 0,C 180,E1 26392.789,E2 26392.789} C_VEL
LIN {X 0,Y 546.546,Z 847.057,A -85,B 0,C 180,E1 26391.35,E2 26391.35} C_VEL
LIN {X 0,Y 545.91,Z 863.371,A -85,B 0,C 180,E1 26389.806,E2 26389.806} C_VEL
LIN {X 0,Y 545.352,Z 878.139,A -85,B 0,C 180,E1 26388.161,E2 26388.161} C_VEL
LIN {X 0,Y 544.901,Z 891.497,A -85,B 0,C 180,E1 26386.414,E2 26386.414} C_VEL
LIN {X 0,Y 544.518,Z 904.116,A -85,B 0,C 180,E1 26384.461,E2 26384.461} C_VEL
LIN {X 0,Y 544.255,Z 915.117,A -85,B 0,C 180,E1 26382.412,E2 26382.412} C_VEL
LIN {X 0,Y 544.08,Z 924.081,A -85,B 0,C 180,E1 26380.375,E2 26380.375} C_VEL
LIN {X 0,Y 543.988,Z 931.236,A -85,B 0,C 180,E1 26378.349,E2 26378.349} C_VEL
LIN {X 0,Y 543.939,Z 936.897,A -85,B 0,C 180,E1 26376.226,E2 26376.226} C_VEL
LIN {X 0,Y 543.919,Z 940.861,A -85,B 0,C 180,E1 26374.111,E2 26374.111} C_VEL
LIN {X 0,Y 543.914,Z 943.278,A -85,B 0,C 180,E1 26371.896,E2 26371.896} C_VEL
LIN {X 0,Y 543.908,Z 943.971,A -85,B 0,C 180,E1 26369.789,E2 26369.789} C_VEL
LIN {X 0,Y 543.906,Z 942.993,A -85,B 0,C 180,E1 26367.577,E2 26367.577} C_VEL
LIN {X 0,Y 543.919,Z 940.2,A -85,B 0,C 180,E1 26365.361,E2 26365.361} C_VEL
LIN {X 0,Y 543.945,Z 935.844,A -85,B 0,C 180,E1 26363.244,E2 26363.244} C_VEL
LIN {X 0,Y 543.998,Z 929.769,A -85,B 0,C 180,E1 26361.118,E2 26361.118} C_VEL
LIN {X 0,Y 544.108,Z 922.29,A -85,B 0,C 180,E1 26359.09,E2 26359.09} C_VEL
LIN {X 0,Y 544.308,Z 912.947,A -85,B 0,C 180,E1 26357.05,E2 26357.05} C_VEL
LIN {X 0,Y 544.604,Z 901.447,A -85,B 0,C 180,E1 26354.997,E2 26354.997} C_VEL
LIN {X 0,Y 544.974,Z 889.035,A -85,B 0,C 180,E1 26353.149,E2 26353.149} C_VEL
LIN {X 0,Y 545.456,Z 875.081,A -85,B 0,C 180,E1 26351.388,E2 26351.388} C_VEL
LIN {X 0,Y 546.032,Z 859.839,A -85,B 0,C 180,E1 26349.752,E2 26349.752} C_VEL
LIN {X 0,Y 546.702,Z 842.819,A -85,B 0,C 180,E1 26348.206,E2 26348.206} C_VEL
LIN {X 0,Y 547.416,Z 824.593,A -85,B 0,C 180,E1 26346.82,E2 26346.82} C_VEL
LIN {X 0,Y 548.089,Z 806.078,A -85,B 0,C 180,E1 26345.651,E2 26345.651} C_VEL
LIN {X 0,Y 548.73,Z 787.808,A -85,B 0,C 180,E1 26344.704,E2 26344.704} C_VEL
LIN {X 0,Y 549.31,Z 768.011,A -85,B 0,C 180,E1 26343.894,E2 26343.894} C_VEL
LIN {X 0,Y 549.767,Z 748.034,A -85,B 0,C 180,E1 26343.277,E2 26343.277} C_VEL
LIN {X 0,Y 550.121,Z 726.999,A -85,B 0,C 180,E1 26342.832,E2 26342.832} C_VEL
LIN {X 0,Y 551.812,Z 480.317,A -85,B 0,C 180,E1 26339.317,E2 26339.317} C_VEL
LIN {X 0,Y 550.131,Z 470.051,A -85,B 0,C 180,E1 26339.046,E2 26339.046} C_VEL
LIN {X 0,Y 551.045,Z 441.347,A -85,B 0,C 180,E1 26337.02,E2 26337.02} C_VEL
LIN {X 0,Y 552.955,Z 399.341,A -85,B 0,C 180,E1 26333.928,E2 26333.928} C_VEL
LIN {X 0,Y 549.226,Z 390.441,A -85,B 0,C 180,E1 26332.88,E2 26332.88} C_VEL
LIN {X 0,Y 545.904,Z 382.988,A -85,B 0,C 180,E1 26331.96,E2 26331.96} C_VEL
LIN {X 0,Y 544.393,Z 379.512,A -85,B 0,C 180,E1 26331.482,E2 26331.482} C_VEL
LIN {X 0,Y 544.349,Z 379.225,A -85,B 0,C 180,E1 26328.699,E2 26328.699} C_VEL
LIN {X 0,Y 544.357,Z 379.223,A -85,B 0,C 180,E1 26325.292,E2 26325.292} C_VEL
LIN {X 0,Y 544.362,Z 379.237,A -85,B 0,C 180,E1 26322.241,E2 26322.241} C_VEL
LIN {X 0,Y 544.347,Z 379.24,A -85,B 0,C 180,E1 26318.848,E2 26318.848} C_VEL
LIN {X 0,Y 544.381,Z 379.217,A -85,B 0,C 180,E1 26315.726,E2 26315.726} C_VEL
LIN {X 0,Y 544.34,Z 379.237,A -85,B 0,C 180,E1 26312.436,E2 26312.436} C_VEL
LIN {X 0,Y 544.405,Z 379.215,A -85,B 0,C 180,E1 26309.245,E2 26309.245} C_VEL
LIN {X 0,Y 544.337,Z 379.235,A -85,B 0,C 180,E1 26306.041,E2 26306.041} C_VEL
LIN {X 0,Y 544.401,Z 379.234,A -85,B 0,C 180,E1 26302.781,E2 26302.781} C_VEL
LIN {X 0,Y 544.337,Z 379.237,A -85,B 0,C 180,E1 26299.558,E2 26299.558} C_VEL
LIN {X 0,Y 544.368,Z 379.237,A -85,B 0,C 180,E1 26296.212,E2 26296.212} C_VEL
LIN {X 0,Y 544.341,Z 379.237,A -85,B 0,C 180,E1 26293.166,E2 26293.166} C_VEL
LIN {X 0,Y 544.347,Z 379.239,A -85,B 0,C 180,E1 26289.729,E2 26289.729} C_VEL
LIN {X 0,Y 544.348,Z 379.232,A -85,B 0,C 180,E1 26286.751,E2 26286.751} C_VEL
LIN {X 0,Y 544.341,Z 379.236,A -85,B 0,C 180,E1 26283.37,E2 26283.37} C_VEL
LIN {X 0,Y 544.374,Z 379.236,A -85,B 0,C 180,E1 26280.211,E2 26280.211} C_VEL
LIN {X 0,Y 544.331,Z 379.237,A -85,B 0,C 180,E1 26276.947,E2 26276.947} C_VEL
LIN {X 0,Y 544.403,Z 379.238,A -85,B 0,C 180,E1 26273.674,E2 26273.674} C_VEL
LIN {X 0,Y 544.327,Z 379.239,A -85,B 0,C 180,E1 26270.485,E2 26270.485} C_VEL
LIN {X 0,Y 544.391,Z 379.215,A -85,B 0,C 180,E1 26267.232,E2 26267.232} C_VEL
LIN {X 0,Y 544.326,Z 379.238,A -85,B 0,C 180,E1 26264.116,E2 26264.116} C_VEL
LIN {X 0,Y 544.37,Z 379.218,A -85,B 0,C 180,E1 26260.806,E2 26260.806} C_VEL
LIN {X 0,Y 544.327,Z 379.239,A -85,B 0,C 180,E1 26257.766,E2 26257.766} C_VEL
LIN {X 0,Y 544.355,Z 379.222,A -85,B 0,C 180,E1 26254.404,E2 26254.404} C_VEL
LIN {X 0,Y 544.332,Z 379.241,A -85,B 0,C 180,E1 26251.353,E2 26251.353} C_VEL
LIN {X 0,Y 544.333,Z 379.241,A -85,B 0,C 180,E1 26247.865,E2 26247.865} C_VEL
LIN {X 0,Y 544.348,Z 379.224,A -85,B 0,C 180,E1 26244.824,E2 26244.824} C_VEL
LIN {X 0,Y 544.324,Z 379.232,A -85,B 0,C 180,E1 26241.487,E2 26241.487} C_VEL
LIN {X 0,Y 544.356,Z 379.233,A -85,B 0,C 180,E1 26238.466,E2 26238.466} C_VEL
LIN {X 0,Y 544.374,Z 379.488,A -85,B 0,C 180,E1 26237.547,E2 26237.547} C_VEL
LIN {X 0,Y 545.17,Z 381.941,A -85,B 0,C 180,E1 26237.267,E2 26237.267} C_VEL
LIN {X 0,Y 546.893,Z 384.873,A -85,B 0,C 180,E1 26236.934,E2 26236.934} C_VEL
LIN {X 0,Y 556.034,Z 401.352,A -85,B 0,C 180,E1 26235.18,E2 26235.18} C_VEL
LIN {X 0,Y 558.191,Z 405.218,A -85,B 0,C 180,E1 26234.784,E2 26234.784} C_VEL
LIN {X 0,Y 556.639,Z 457.878,A -85,B 0,C 180,E1 26231.958,E2 26231.958} C_VEL
LIN {X 0,Y 556.601,Z 466.61,A -85,B 0,C 180,E1 26231.524,E2 26231.524} C_VEL
LIN {X 0,Y 558.061,Z 478.548,A -85,B 0,C 180,E1 26231.192,E2 26231.192} C_VEL
LIN {X 0,Y 556.036,Z 682.751,A -85,B 0,C 180,E1 26228.016,E2 26228.016} C_VEL
LIN {X 0,Y 554.725,Z 816.214,A -85,B 0,C 180,E1 26225.966,E2 26225.966} C_VEL
LIN {X 0,Y 554.106,Z 839.741,A -85,B 0,C 180,E1 26225.417,E2 26225.417} C_VEL
LIN {X 0,Y 553.43,Z 861.714,A -85,B 0,C 180,E1 26224.716,E2 26224.716} C_VEL
LIN {X 0,Y 552.558,Z 883.675,A -85,B 0,C 180,E1 26223.809,E2 26223.809} C_VEL
LIN {X 0,Y 551.622,Z 904.867,A -85,B 0,C 180,E1 26222.751,E2 26222.751} C_VEL
LIN {X 0,Y 550.592,Z 925.939,A -85,B 0,C 180,E1 26221.473,E2 26221.473} C_VEL
LIN {X 0,Y 549.502,Z 946.824,A -85,B 0,C 180,E1 26219.991,E2 26219.991} C_VEL
LIN {X 0,Y 548.553,Z 965.252,A -85,B 0,C 180,E1 26218.467,E2 26218.467} C_VEL
LIN {X 0,Y 547.543,Z 984.455,A -85,B 0,C 180,E1 26216.635,E2 26216.635} C_VEL
LIN {X 0,Y 546.691,Z 1001.616,A -85,B 0,C 180,E1 26214.761,E2 26214.761} C_VEL
LIN {X 0,Y 545.969,Z 1016.841,A -85,B 0,C 180,E1 26212.846,E2 26212.846} C_VEL
LIN {X 0,Y 545.304,Z 1032.339,A -85,B 0,C 180,E1 26210.613,E2 26210.613} C_VEL
LIN {X 0,Y 544.835,Z 1045.002,A -85,B 0,C 180,E1 26208.511,E2 26208.511} C_VEL
LIN {X 0,Y 544.476,Z 1056.321,A -85,B 0,C 180,E1 26206.318,E2 26206.318} C_VEL
LIN {X 0,Y 544.23,Z 1066.336,A -85,B 0,C 180,E1 26204.062,E2 26204.062} C_VEL
LIN {X 0,Y 544.073,Z 1074.698,A -85,B 0,C 180,E1 26201.77,E2 26201.77} C_VEL
LIN {X 0,Y 543.965,Z 1081.774,A -85,B 0,C 180,E1 26199.415,E2 26199.415} C_VEL
LIN {X 0,Y 543.904,Z 1086.841,A -85,B 0,C 180,E1 26197.181,E2 26197.181} C_VEL
LIN {X 0,Y 543.913,Z 1090.436,A -85,B 0,C 180,E1 26195.062,E2 26195.062} C_VEL
LIN {X 0,Y 543.912,Z 1093.055,A -85,B 0,C 180,E1 26192.529,E2 26192.529} C_VEL
LIN {X 0,Y 543.892,Z 1093.939,A -85,B 0,C 180,E1 26190.316,E2 26190.316} C_VEL
LIN {X 0,Y 543.913,Z 1093.324,A -85,B 0,C 180,E1 26187.893,E2 26187.893} C_VEL
LIN {X 0,Y 543.912,Z 1091.389,A -85,B 0,C 180,E1 26185.678,E2 26185.678} C_VEL
LIN {X 0,Y 543.913,Z 1087.667,A -85,B 0,C 180,E1 26183.243,E2 26183.243} C_VEL
LIN {X 0,Y 543.966,Z 1083.061,A -85,B 0,C 180,E1 26181.118,E2 26181.118} C_VEL
LIN {X 0,Y 544.038,Z 1076.118,A -85,B 0,C 180,E1 26178.659,E2 26178.659} C_VEL
LIN {X 0,Y 544.169,Z 1068.52,A -85,B 0,C 180,E1 26176.505,E2 26176.505} C_VEL
LIN {X 0,Y 544.418,Z 1058.399,A -85,B 0,C 180,E1 26174.118,E2 26174.118} C_VEL
LIN {X 0,Y 544.746,Z 1047.983,A -85,B 0,C 180,E1 26172.04,E2 26172.04} C_VEL
LIN {X 0,Y 545.236,Z 1034.464,A -85,B 0,C 180,E1 26169.721,E2 26169.721} C_VEL
LIN {X 0,Y 545.84,Z 1020.216,A -85,B 0,C 180,E1 26167.603,E2 26167.603} C_VEL
LIN {X 0,Y 546.545,Z 1004.407,A -85,B 0,C 180,E1 26165.578,E2 26165.578} C_VEL
LIN {X 0,Y 547.465,Z 986.115,A -85,B 0,C 180,E1 26163.536,E2 26163.536} C_VEL
LIN {X 0,Y 548.428,Z 967.896,A -85,B 0,C 180,E1 26161.764,E2 26161.764} C_VEL
LIN {X 0,Y 549.412,Z 948.596,A -85,B 0,C 180,E1 26160.149,E2 26160.149} C_VEL
LIN {X 0,Y 550.535,Z 927.112,A -85,B 0,C 180,E1 26158.604,E2 26158.604} C_VEL
LIN {X 0,Y 551.474,Z 907.816,A -85,B 0,C 180,E1 26157.419,E2 26157.419} C_VEL
LIN {X 0,Y 552.44,Z 886.233,A -85,B 0,C 180,E1 26156.307,E2 26156.307} C_VEL
LIN {X 0,Y 553.256,Z 866.434,A -85,B 0,C 180,E1 26155.466,E2 26155.466} C_VEL
LIN {X 0,Y 554.003,Z 842.948,A -85,B 0,C 180,E1 26154.673,E2 26154.673} C_VEL
LIN {X 0,Y 554.617,Z 821.095,A -85,B 0,C 180,E1 26154.129,E2 26154.129} C_VEL
LIN {X 0,Y 555.064,Z 787.339,A -85,B 0,C 180,E1 26153.571,E2 26153.571} C_VEL
LIN {X 0,Y 557.029,Z 579.661,A -85,B 0,C 180,E1 26150.393,E2 26150.393} C_VEL
LIN {X 0,Y 557.922,Z 475.965,A -85,B 0,C 180,E1 26148.753,E2 26148.753} C_VEL
LIN {X 0,Y 556.457,Z 464.889,A -85,B 0,C 180,E1 26148.411,E2 26148.411} C_VEL
LIN {X 0,Y 558.142,Z 408.591,A -85,B 0,C 180,E1 26145.393,E2 26145.393} C_VEL
LIN {X 0,Y 558.101,Z 404.872,A -85,B 0,C 180,E1 26145.19,E2 26145.19} C_VEL
LIN {X 0,Y 549.078,Z 388.844,A -85,B 0,C 180,E1 26143.497,E2 26143.497} C_VEL
LIN {X 0,Y 545.665,Z 382.766,A -85,B 0,C 180,E1 26142.828,E2 26142.828} C_VEL
LIN {X 0,Y 544.408,Z 379.693,A -85,B 0,C 180,E1 26142.485,E2 26142.485} C_VEL
LIN {X 0,Y 544.376,Z 379.217,A -85,B 0,C 180,E1 26142.095,E2 26142.095} C_VEL
LIN {X 0,Y 544.318,Z 379.228,A -85,B 0,C 180,E1 26138.844,E2 26138.844} C_VEL
LIN {X 0,Y 544.386,Z 379.22,A -85,B 0,C 180,E1 26135.726,E2 26135.726} C_VEL
LIN {X 0,Y 544.321,Z 379.241,A -85,B 0,C 180,E1 26132.527,E2 26132.527} C_VEL
LIN {X 0,Y 544.393,Z 379.231,A -85,B 0,C 180,E1 26129.245,E2 26129.245} C_VEL
LIN {X 0,Y 544.323,Z 379.229,A -85,B 0,C 180,E1 26126.041,E2 26126.041} C_VEL
LIN {X 0,Y 544.357,Z 379.239,A -85,B 0,C 180,E1 26122.688,E2 26122.688} C_VEL
LIN {X 0,Y 544.329,Z 379.221,A -85,B 0,C 180,E1 26119.642,E2 26119.642} C_VEL
LIN {X 0,Y 544.34,Z 379.238,A -85,B 0,C 180,E1 26116.212,E2 26116.212} C_VEL
LIN {X 0,Y 544.339,Z 379.221,A -85,B 0,C 180,E1 26113.213,E2 26113.213} C_VEL
LIN {X 0,Y 544.334,Z 379.237,A -85,B 0,C 180,E1 26109.836,E2 26109.836} C_VEL
LIN {X 0,Y 544.348,Z 379.234,A -85,B 0,C 180,E1 26106.857,E2 26106.857} C_VEL
LIN {X 0,Y 544.331,Z 379.236,A -85,B 0,C 180,E1 26103.475,E2 26103.475} C_VEL
LIN {X 0,Y 544.379,Z 379.234,A -85,B 0,C 180,E1 26100.315,E2 26100.315} C_VEL
LIN {X 0,Y 544.327,Z 379.236,A -85,B 0,C 180,E1 26097.052,E2 26097.052} C_VEL
LIN {X 0,Y 544.404,Z 379.233,A -85,B 0,C 180,E1 26093.779,E2 26093.779} C_VEL
LIN {X 0,Y 544.33,Z 379.239,A -85,B 0,C 180,E1 26090.541,E2 26090.541} C_VEL
LIN {X 0,Y 544.374,Z 379.237,A -85,B 0,C 180,E1 26087.24,E2 26087.24} C_VEL
LIN {X 0,Y 544.332,Z 379.236,A -85,B 0,C 180,E1 26084.225,E2 26084.225} C_VEL
LIN {X 0,Y 544.369,Z 379.237,A -85,B 0,C 180,E1 26080.917,E2 26080.917} C_VEL
LIN {X 0,Y 544.334,Z 379.235,A -85,B 0,C 180,E1 26077.879,E2 26077.879} C_VEL
LIN {X 0,Y 544.361,Z 379.235,A -85,B 0,C 180,E1 26074.545,E2 26074.545} C_VEL
LIN {X 0,Y 544.344,Z 379.238,A -85,B 0,C 180,E1 26071.473,E2 26071.473} C_VEL
LIN {X 0,Y 544.356,Z 379.218,A -85,B 0,C 180,E1 26069.211,E2 26069.211} C_VEL
LIN {X 0,Y 543.414,Z 379.352,A -85,B 0,C 180,E1 26068.4,E2 26068.4} C_VEL
LIN {X 0,Y 536.837,Z 380.173,A -85,B 0,C 180,E1 26066.064,E2 26066.064} C_VEL
LIN {X 0,Y 536.395,Z 380.225,A -85,B 0,C 180,E1 26065.529,E2 26065.529} C_VEL
LIN {X 0,Y 536.443,Z 380.226,A -85,B 0,C 180,E1 26062.177,E2 26062.177} C_VEL
LIN {X 0,Y 536.402,Z 380.211,A -85,B 0,C 180,E1 26059.019,E2 26059.019} C_VEL
LIN {X 0,Y 536.406,Z 380.22,A -85,B 0,C 180,E1 26055.503,E2 26055.503} C_VEL
LIN {X 0,Y 536.441,Z 380.226,A -85,B 0,C 180,E1 26052.289,E2 26052.289} C_VEL
LIN {X 0,Y 536.426,Z 380.372,A -85,B 0,C 180,E1 26049.189,E2 26049.189} C_VEL
LIN {X 0,Y 536.964,Z 382.351,A -85,B 0,C 180,E1 26048.891,E2 26048.891} C_VEL
LIN {X 0,Y 540.359,Z 389.199,A -85,B 0,C 180,E1 26047.977,E2 26047.977} C_VEL
LIN {X 0,Y 546.275,Z 402.842,A -85,B 0,C 180,E1 26046.307,E2 26046.307} C_VEL
LIN {X 0,Y 544.326,Z 443.249,A -85,B 0,C 180,E1 26043.303,E2 26043.303} C_VEL
LIN {X 0,Y 543.23,Z 470.598,A -85,B 0,C 180,E1 26041.326,E2 26041.326} C_VEL
LIN {X 0,Y 544.952,Z 483.076,A -85,B 0,C 180,E1 26040.984,E2 26040.984} C_VEL
LIN {X 0,Y 542.951,Z 732.549,A -85,B 0,C 180,E1 26037.369,E2 26037.369} C_VEL
LIN {X 0,Y 542.481,Z 753.386,A -85,B 0,C 180,E1 26036.868,E2 26036.868} C_VEL
LIN {X 0,Y 541.904,Z 773.123,A -85,B 0,C 180,E1 26036.196,E2 26036.196} C_VEL
LIN {X 0,Y 541.229,Z 792.861,A -85,B 0,C 180,E1 26035.32,E2 26035.32} C_VEL
LIN {X 0,Y 540.48,Z 811.392,A -85,B 0,C 180,E1 26034.296,E2 26034.296} C_VEL
LIN {X 0,Y 539.72,Z 829.593,A -85,B 0,C 180,E1 26033.074,E2 26033.074} C_VEL
LIN {X 0,Y 538.939,Z 847.285,A -85,B 0,C 180,E1 26031.647,E2 26031.647} C_VEL
LIN {X 0,Y 538.199,Z 863.931,A -85,B 0,C 180,E1 26030.045,E2 26030.045} C_VEL
LIN {X 0,Y 537.545,Z 879.069,A -85,B 0,C 180,E1 26028.322,E2 26028.322} C_VEL
LIN {X 0,Y 537.031,Z 892.271,A -85,B 0,C 180,E1 26026.551,E2 26026.551} C_VEL
LIN {X 0,Y 536.618,Z 904.119,A -85,B 0,C 180,E1 26024.679,E2 26024.679} C_VEL
LIN {X 0,Y 536.311,Z 915.122,A -85,B 0,C 180,E1 26022.599,E2 26022.599} C_VEL
LIN {X 0,Y 536.113,Z 924.084,A -85,B 0,C 180,E1 26020.531,E2 26020.531} C_VEL
LIN {X 0,Y 536.004,Z 931.239,A -85,B 0,C 180,E1 26018.474,E2 26018.474} C_VEL
LIN {X 0,Y 535.944,Z 936.899,A -85,B 0,C 180,E1 26016.319,E2 26016.319} C_VEL
LIN {X 0,Y 535.921,Z 940.863,A -85,B 0,C 180,E1 26014.173,E2 26014.173} C_VEL
LIN {X 0,Y 535.914,Z 943.278,A -85,B 0,C 180,E1 26011.925,E2 26011.925} C_VEL
LIN {X 0,Y 535.909,Z 943.971,A -85,B 0,C 180,E1 26009.786,E2 26009.786} C_VEL
LIN {X 0,Y 535.906,Z 942.992,A -85,B 0,C 180,E1 26007.541,E2 26007.541} C_VEL
LIN {X 0,Y 535.921,Z 940.198,A -85,B 0,C 180,E1 26005.291,E2 26005.291} C_VEL
LIN {X 0,Y 535.949,Z 935.842,A -85,B 0,C 180,E1 26003.143,E2 26003.143} C_VEL
LIN {X 0,Y 536.01,Z 929.767,A -85,B 0,C 180,E1 26000.985,E2 26000.985} C_VEL
LIN {X 0,Y 536.142,Z 922.286,A -85,B 0,C 180,E1 25998.925,E2 25998.925} C_VEL
LIN {X 0,Y 536.373,Z 912.943,A -85,B 0,C 180,E1 25996.855,E2 25996.855} C_VEL
LIN {X 0,Y 536.719,Z 901.444,A -85,B 0,C 180,E1 25994.771,E2 25994.771} C_VEL
LIN {X 0,Y 537.146,Z 889.031,A -85,B 0,C 180,E1 25992.896,E2 25992.896} C_VEL
LIN {X 0,Y 537.696,Z 875.179,A -85,B 0,C 180,E1 25991.122,E2 25991.122} C_VEL
LIN {X 0,Y 538.354,Z 859.83,A -85,B 0,C 180,E1 25989.45,E2 25989.45} C_VEL
LIN {X 0,Y 539.117,Z 842.808,A -85,B 0,C 180,E1 25987.884,E2 25987.884} C_VEL
LIN {X 0,Y 539.904,Z 825.392,A -85,B 0,C 180,E1 25986.536,E2 25986.536} C_VEL
LIN {X 0,Y 540.669,Z 807.064,A -85,B 0,C 180,E1 25985.353,E2 25985.353} C_VEL
LIN {X 0,Y 541.414,Z 788.118,A -85,B 0,C 180,E1 25984.354,E2 25984.354} C_VEL
LIN {X 0,Y 542.056,Z 768.73,A -85,B 0,C 180,E1 25983.547,E2 25983.547} C_VEL
LIN {X 0,Y 542.587,Z 748.619,A -85,B 0,C 180,E1 25982.912,E2 25982.912} C_VEL
LIN {X 0,Y 542.995,Z 727.381,A -85,B 0,C 180,E1 25982.453,E2 25982.453} C_VEL
LIN {X 0,Y 544.934,Z 481.522,A -85,B 0,C 180,E1 25978.899,E2 25978.899} C_VEL
LIN {X 0,Y 543.166,Z 469.708,A -85,B 0,C 180,E1 25978.542,E2 25978.542} C_VEL
LIN {X 0,Y 545.355,Z 421.923,A -85,B 0,C 180,E1 25975.039,E2 25975.039} C_VEL
LIN {X 0,Y 546.2,Z 402.581,A -85,B 0,C 180,E1 25973.575,E2 25973.575} C_VEL
LIN {X 0,Y 539.752,Z 387.856,A -85,B 0,C 180,E1 25971.761,E2 25971.761} C_VEL
LIN {X 0,Y 536.476,Z 380.649,A -85,B 0,C 180,E1 25970.798,E2 25970.798} C_VEL
LIN {X 0,Y 536.443,Z 380.216,A -85,B 0,C 180,E1 25970.398,E2 25970.398} C_VEL
LIN {X 0,Y 536.407,Z 380.23,A -85,B 0,C 180,E1 25967.101,E2 25967.101} C_VEL
LIN {X 0,Y 536.465,Z 380.219,A -85,B 0,C 180,E1 25963.839,E2 25963.839} C_VEL
LIN {X 0,Y 536.4,Z 380.213,A -85,B 0,C 180,E1 25960.583,E2 25960.583} C_VEL
LIN {X 0,Y 536.449,Z 380.215,A -85,B 0,C 180,E1 25957.283,E2 25957.283} C_VEL
LIN {X 0,Y 536.405,Z 380.224,A -85,B 0,C 180,E1 25954.13,E2 25954.13} C_VEL
LIN {X 0,Y 536.418,Z 380.204,A -85,B 0,C 180,E1 25950.712,E2 25950.712} C_VEL
LIN {X 0,Y 536.414,Z 380.224,A -85,B 0,C 180,E1 25947.654,E2 25947.654} C_VEL
LIN {X 0,Y 536.404,Z 380.228,A -85,B 0,C 180,E1 25944.21,E2 25944.21} C_VEL
LIN {X 0,Y 536.458,Z 380.221,A -85,B 0,C 180,E1 25940.968,E2 25940.968} C_VEL
LIN {X 0,Y 536.396,Z 380.226,A -85,B 0,C 180,E1 25937.689,E2 25937.689} C_VEL
LIN {X 0,Y 536.467,Z 380.22,A -85,B 0,C 180,E1 25934.463,E2 25934.463} C_VEL
LIN {X 0,Y 536.394,Z 380.221,A -85,B 0,C 180,E1 25931.287,E2 25931.287} C_VEL
LIN {X 0,Y 536.448,Z 380.222,A -85,B 0,C 180,E1 25928.036,E2 25928.036} C_VEL
LIN {X 0,Y 536.395,Z 380.227,A -85,B 0,C 180,E1 25924.919,E2 25924.919} C_VEL
LIN {X 0,Y 536.417,Z 380.228,A -85,B 0,C 180,E1 25921.496,E2 25921.496} C_VEL
LIN {X 0,Y 536.4,Z 380.225,A -85,B 0,C 180,E1 25918.505,E2 25918.505} C_VEL
LIN {X 0,Y 536.397,Z 380.228,A -85,B 0,C 180,E1 25914.974,E2 25914.974} C_VEL
LIN {X 0,Y 536.419,Z 380.221,A -85,B 0,C 180,E1 25911.964,E2 25911.964} C_VEL
LIN {X 0,Y 536.39,Z 380.218,A -85,B 0,C 180,E1 25908.604,E2 25908.604} C_VEL
LIN {X 0,Y 536.465,Z 380.21,A -85,B 0,C 180,E1 25905.311,E2 25905.311} C_VEL
LIN {X 0,Y 536.387,Z 380.222,A -85,B 0,C 180,E1 25902.088,E2 25902.088} C_VEL
LIN {X 0,Y 536.435,Z 380.219,A -85,B 0,C 180,E1 25898.742,E2 25898.742} C_VEL
LIN {X 0,Y 536.388,Z 380.222,A -85,B 0,C 180,E1 25895.673,E2 25895.673} C_VEL
LIN {X 0,Y 536.416,Z 380.231,A -85,B 0,C 180,E1 25892.299,E2 25892.299} C_VEL
LIN {X 0,Y 536.392,Z 380.209,A -85,B 0,C 180,E1 25889.242,E2 25889.242} C_VEL
LIN {X 0,Y 536.391,Z 380.221,A -85,B 0,C 180,E1 25885.741,E2 25885.741} C_VEL
LIN {X 0,Y 536.428,Z 380.231,A -85,B 0,C 180,E1 25882.564,E2 25882.564} C_VEL
LIN {X 0,Y 536.382,Z 380.23,A -85,B 0,C 180,E1 25879.276,E2 25879.276} C_VEL
LIN {X 0,Y 536.469,Z 380.443,A -85,B 0,C 180,E1 25878.29,E2 25878.29} C_VEL
LIN {X 0,Y 536.992,Z 382.258,A -85,B 0,C 180,E1 25878.053,E2 25878.053} C_VEL
LIN {X 0,Y 539.11,Z 386.175,A -85,B 0,C 180,E1 25877.611,E2 25877.611} C_VEL
LIN {X 0,Y 551.742,Z 409.037,A -85,B 0,C 180,E1 25875.136,E2 25875.136} C_VEL
LIN {X 0,Y 550.746,Z 450.317,A -85,B 0,C 180,E1 25872.944,E2 25872.944} C_VEL
LIN {X 0,Y 550.35,Z 466.405,A -85,B 0,C 180,E1 25872.107,E2 25872.107} C_VEL
LIN {X 0,Y 552.024,Z 479.916,A -85,B 0,C 180,E1 25871.719,E2 25871.719} C_VEL
LIN {X 0,Y 549.72,Z 684,A -85,B 0,C 180,E1 25868.512,E2 25868.512} C_VEL
LIN {X 0,Y 548.242,Z 816.309,A -85,B 0,C 180,E1 25866.458,E2 25866.458} C_VEL
LIN {X 0,Y 547.56,Z 839.74,A -85,B 0,C 180,E1 25865.905,E2 25865.905} C_VEL
LIN {X 0,Y 546.781,Z 861.599,A -85,B 0,C 180,E1 25865.204,E2 25865.204} C_VEL
LIN {X 0,Y 545.868,Z 882.389,A -85,B 0,C 180,E1 25864.344,E2 25864.344} C_VEL
LIN {X 0,Y 544.922,Z 901.443,A -85,B 0,C 180,E1 25863.399,E2 25863.399} C_VEL
LIN {X 0,Y 543.72,Z 923.243,A -85,B 0,C 180,E1 25862.104,E2 25862.104} C_VEL
LIN {X 0,Y 542.584,Z 943.402,A -85,B 0,C 180,E1 25860.694,E2 25860.694} C_VEL
LIN {X 0,Y 541.366,Z 963.269,A -85,B 0,C 180,E1 25859.061,E2 25859.061} C_VEL
LIN {X 0,Y 540.204,Z 982.789,A -85,B 0,C 180,E1 25857.205,E2 25857.205} C_VEL
LIN {X 0,Y 539.248,Z 999.659,A -85,B 0,C 180,E1 25855.361,E2 25855.361} C_VEL
LIN {X 0,Y 538.34,Z 1015.994,A -85,B 0,C 180,E1 25853.304,E2 25853.304} C_VEL
LIN {X 0,Y 537.604,Z 1030.923,A -85,B 0,C 180,E1 25851.15,E2 25851.15} C_VEL
LIN {X 0,Y 537.052,Z 1043.73,A -85,B 0,C 180,E1 25849.015,E2 25849.015} C_VEL
LIN {X 0,Y 536.601,Z 1055.801,A -85,B 0,C 180,E1 25846.676,E2 25846.676} C_VEL
LIN {X 0,Y 536.315,Z 1065.533,A -85,B 0,C 180,E1 25844.467,E2 25844.467} C_VEL
LIN {X 0,Y 536.101,Z 1074.343,A -85,B 0,C 180,E1 25842.057,E2 25842.057} C_VEL
LIN {X 0,Y 535.976,Z 1080.868,A -85,B 0,C 180,E1 25839.882,E2 25839.882} C_VEL
LIN {X 0,Y 535.917,Z 1086.634,A -85,B 0,C 180,E1 25837.396,E2 25837.396} C_VEL
LIN {X 0,Y 535.914,Z 1090.277,A -85,B 0,C 180,E1 25835.245,E2 25835.245} C_VEL
LIN {X 0,Y 535.898,Z 1092.92,A -85,B 0,C 180,E1 25832.781,E2 25832.781} C_VEL
LIN {X 0,Y 535.884,Z 1093.872,A -85,B 0,C 180,E1 25830.641,E2 25830.641} C_VEL
LIN {X 0,Y 535.906,Z 1093.526,A -85,B 0,C 180,E1 25828.182,E2 25828.182} C_VEL
LIN {X 0,Y 535.916,Z 1091.616,A -85,B 0,C 180,E1 25825.827,E2 25825.827} C_VEL
LIN {X 0,Y 535.922,Z 1088.08,A -85,B 0,C 180,E1 25823.358,E2 25823.358} C_VEL
LIN {X 0,Y 535.969,Z 1083.572,A -85,B 0,C 180,E1 25821.201,E2 25821.201} C_VEL
LIN {X 0,Y 536.045,Z 1077.177,A -85,B 0,C 180,E1 25818.814,E2 25818.814} C_VEL
LIN {X 0,Y 536.197,Z 1069.339,A -85,B 0,C 180,E1 25816.521,E2 25816.521} C_VEL
LIN {X 0,Y 536.469,Z 1059.941,A -85,B 0,C 180,E1 25814.21,E2 25814.21} C_VEL
LIN {X 0,Y 536.84,Z 1049.146,A -85,B 0,C 180,E1 25811.99,E2 25811.99} C_VEL
LIN {X 0,Y 537.393,Z 1035.863,A -85,B 0,C 180,E1 25809.639,E2 25809.639} C_VEL
LIN {X 0,Y 538.014,Z 1022.559,A -85,B 0,C 180,E1 25807.606,E2 25807.606} C_VEL
LIN {X 0,Y 538.862,Z 1006.266,A -85,B 0,C 180,E1 25805.441,E2 25805.441} C_VEL
LIN {X 0,Y 539.841,Z 989.433,A -85,B 0,C 180,E1 25803.489,E2 25803.489} C_VEL
LIN {X 0,Y 540.864,Z 971.573,A -85,B 0,C 180,E1 25801.694,E2 25801.694} C_VEL
LIN {X 0,Y 542.072,Z 951.525,A -85,B 0,C 180,E1 25799.948,E2 25799.948} C_VEL
LIN {X 0,Y 543.279,Z 931.482,A -85,B 0,C 180,E1 25798.441,E2 25798.441} C_VEL
LIN {X 0,Y 544.416,Z 910.827,A -85,B 0,C 180,E1 25797.132,E2 25797.132} C_VEL
LIN {X 0,Y 545.496,Z 890.053,A -85,B 0,C 180,E1 25796.01,E2 25796.01} C_VEL
LIN {X 0,Y 546.46,Z 869.192,A -85,B 0,C 180,E1 25795.093,E2 25795.093} C_VEL
LIN {X 0,Y 547.346,Z 847.02,A -85,B 0,C 180,E1 25794.305,E2 25794.305} C_VEL
LIN {X 0,Y 547.977,Z 824.991,A -85,B 0,C 180,E1 25793.722,E2 25793.722} C_VEL
LIN {X 0,Y 548.524,Z 797.645,A -85,B 0,C 180,E1 25793.23,E2 25793.23} C_VEL
LIN {X 0,Y 550.797,Z 586.29,A -85,B 0,C 180,E1 25789.966,E2 25789.966} C_VEL
LIN {X 0,Y 551.877,Z 477.357,A -85,B 0,C 180,E1 25788.224,E2 25788.224} C_VEL
LIN {X 0,Y 550.238,Z 464.635,A -85,B 0,C 180,E1 25787.822,E2 25787.822} C_VEL
LIN {X 0,Y 551.435,Z 424.585,A -85,B 0,C 180,E1 25785.686,E2 25785.686} C_VEL
LIN {X 0,Y 551.625,Z 408.722,A -85,B 0,C 180,E1 25784.836,E2 25784.836} C_VEL
LIN {X 0,Y 543.425,Z 394.076,A -85,B 0,C 180,E1 25783.264,E2 25783.264} C_VEL
LIN {X 0,Y 537.937,Z 383.976,A -85,B 0,C 180,E1 25782.143,E2 25782.143} C_VEL
LIN {X 0,Y 536.502,Z 380.61,A -85,B 0,C 180,E1 25781.746,E2 25781.746} C_VEL
LIN {X 0,Y 536.396,Z 380.229,A -85,B 0,C 180,E1 25781.289,E2 25781.289} C_VEL
LIN {X 0,Y 536.402,Z 380.221,A -85,B 0,C 180,E1 25778.232,E2 25778.232} C_VEL
LIN {X 0,Y 536.388,Z 380.215,A -85,B 0,C 180,E1 25774.896,E2 25774.896} C_VEL
LIN {X 0,Y 536.421,Z 380.217,A -85,B 0,C 180,E1 25771.792,E2 25771.792} C_VEL
LIN {X 0,Y 536.386,Z 380.23,A -85,B 0,C 180,E1 25768.502,E2 25768.502} C_VEL
LIN {X 0,Y 536.444,Z 380.206,A -85,B 0,C 180,E1 25765.313,E2 25765.313} C_VEL
LIN {X 0,Y 536.385,Z 380.229,A -85,B 0,C 180,E1 25762.112,E2 25762.112} C_VEL
LIN {X 0,Y 536.454,Z 380.204,A -85,B 0,C 180,E1 25758.923,E2 25758.923} C_VEL
LIN {X 0,Y 536.386,Z 380.228,A -85,B 0,C 180,E1 25755.681,E2 25755.681} C_VEL
LIN {X 0,Y 536.437,Z 380.205,A -85,B 0,C 180,E1 25752.396,E2 25752.396} C_VEL
LIN {X 0,Y 536.392,Z 380.227,A -85,B 0,C 180,E1 25749.224,E2 25749.224} C_VEL
LIN {X 0,Y 536.404,Z 380.226,A -85,B 0,C 180,E1 25745.777,E2 25745.777} C_VEL
LIN {X 0,Y 536.412,Z 380.226,A -85,B 0,C 180,E1 25742.671,E2 25742.671} C_VEL
LIN {X 0,Y 536.391,Z 380.227,A -85,B 0,C 180,E1 25739.252,E2 25739.252} C_VEL
LIN {X 0,Y 536.45,Z 380.222,A -85,B 0,C 180,E1 25736.045,E2 25736.045} C_VEL
LIN {X 0,Y 536.388,Z 380.222,A -85,B 0,C 180,E1 25732.825,E2 25732.825} C_VEL
LIN {X 0,Y 536.459,Z 380.22,A -85,B 0,C 180,E1 25729.584,E2 25729.584} C_VEL
LIN {X 0,Y 536.39,Z 380.228,A -85,B 0,C 180,E1 25726.416,E2 25726.416} C_VEL
LIN {X 0,Y 536.454,Z 380.225,A -85,B 0,C 180,E1 25723.208,E2 25723.208} C_VEL
LIN {X 0,Y 536.398,Z 380.228,A -85,B 0,C 180,E1 25719.941,E2 25719.941} C_VEL
LIN {X 0,Y 536.408,Z 380.227,A -85,B 0,C 180,E1 25716.491,E2 25716.491} C_VEL
LIN {X 0,Y 536.415,Z 380.226,A -85,B 0,C 180,E1 25713.426,E2 25713.426} C_VEL
LIN {X 0,Y 536.395,Z 380.205,A -85,B 0,C 180,E1 25710.029,E2 25710.029} C_VEL
LIN {X 0,Y 536.443,Z 380.228,A -85,B 0,C 180,E1 25706.899,E2 25706.899} C_VEL
LIN {X 0,Y 536.395,Z 380.225,A -85,B 0,C 180,E1 25705.529,E2 25705.529} C_VEL
LIN {X 0,Y 535.421,Z 380.35,A -85,B 0,C 180,E1 25704.706,E2 25704.706} C_VEL
LIN {X 0,Y 528.93,Z 381.163,A -85,B 0,C 180,E1 25702.335,E2 25702.335} C_VEL
LIN {X 0,Y 528.469,Z 381.218,A -85,B 0,C 180,E1 25701.792,E2 25701.792} C_VEL
LIN {X 0,Y 528.486,Z 381.195,A -85,B 0,C 180,E1 25698.678,E2 25698.678} C_VEL
LIN {X 0,Y 528.46,Z 381.206,A -85,B 0,C 180,E1 25695.35,E2 25695.35} C_VEL
LIN {X 0,Y 528.515,Z 381.209,A -85,B 0,C 180,E1 25692.132,E2 25692.132} C_VEL
LIN {X 0,Y 528.54,Z 381.306,A -85,B 0,C 180,E1 25689.949,E2 25689.949} C_VEL
LIN {X 0,Y 528.872,Z 382.769,A -85,B 0,C 180,E1 25689.695,E2 25689.695} C_VEL
LIN {X 0,Y 535.885,Z 397.689,A -85,B 0,C 180,E1 25687.711,E2 25687.711} C_VEL
LIN {X 0,Y 539.679,Z 406.459,A -85,B 0,C 180,E1 25686.625,E2 25686.625} C_VEL
LIN {X 0,Y 537.431,Z 449.272,A -85,B 0,C 180,E1 25683.415,E2 25683.415} C_VEL
LIN {X 0,Y 536.528,Z 470.556,A -85,B 0,C 180,E1 25681.868,E2 25681.868} C_VEL
LIN {X 0,Y 538.574,Z 484.332,A -85,B 0,C 180,E1 25681.482,E2 25681.482} C_VEL
LIN {X 0,Y 536.345,Z 680.743,A -85,B 0,C 180,E1 25678.538,E2 25678.538} C_VEL
LIN {X 0,Y 535.824,Z 733.558,A -85,B 0,C 180,E1 25677.744,E2 25677.744} C_VEL
LIN {X 0,Y 535.303,Z 754.621,A -85,B 0,C 180,E1 25677.223,E2 25677.223} C_VEL
LIN {X 0,Y 534.634,Z 774.616,A -85,B 0,C 180,E1 25676.52,E2 25676.52} C_VEL
LIN {X 0,Y 533.88,Z 794.001,A -85,B 0,C 180,E1 25675.634,E2 25675.634} C_VEL
LIN {X 0,Y 532.987,Z 813.588,A -85,B 0,C 180,E1 25674.517,E2 25674.517} C_VEL
LIN {X 0,Y 532.106,Z 831.902,A -85,B 0,C 180,E1 25673.239,E2 25673.239} C_VEL
LIN {X 0,Y 531.262,Z 848.918,A -85,B 0,C 180,E1 25671.821,E2 25671.821} C_VEL
LIN {X 0,Y 530.469,Z 865.003,A -85,B 0,C 180,E1 25670.235,E2 25670.235} C_VEL
LIN {X 0,Y 529.743,Z 879.999,A -85,B 0,C 180,E1 25668.487,E2 25668.487} C_VEL
LIN {X 0,Y 529.137,Z 893.814,A -85,B 0,C 180,E1 25666.579,E2 25666.579} C_VEL
LIN {X 0,Y 528.68,Z 905.393,A -85,B 0,C 180,E1 25664.68,E2 25664.68} C_VEL
LIN {X 0,Y 528.356,Z 915.64,A -85,B 0,C 180,E1 25662.681,E2 25662.681} C_VEL
LIN {X 0,Y 528.135,Z 924.494,A -85,B 0,C 180,E1 25660.582,E2 25660.582} C_VEL
LIN {X 0,Y 528.013,Z 931.565,A -85,B 0,C 180,E1 25658.494,E2 25658.494} C_VEL
LIN {X 0,Y 527.944,Z 937.408,A -85,B 0,C 180,E1 25656.197,E2 25656.197} C_VEL
LIN {X 0,Y 527.919,Z 941.18,A -85,B 0,C 180,E1 25654.018,E2 25654.018} C_VEL
LIN {X 0,Y 527.912,Z 943.346,A -85,B 0,C 180,E1 25651.845,E2 25651.845} C_VEL
LIN {X 0,Y 527.903,Z 943.949,A -85,B 0,C 180,E1 25649.674,E2 25649.674} C_VEL
LIN {X 0,Y 527.906,Z 942.992,A -85,B 0,C 180,E1 25647.503,E2 25647.503} C_VEL
LIN {X 0,Y 527.921,Z 940.356,A -85,B 0,C 180,E1 25645.329,E2 25645.329} C_VEL
LIN {X 0,Y 527.953,Z 936.094,A -85,B 0,C 180,E1 25643.148,E2 25643.148} C_VEL
LIN {X 0,Y 528.022,Z 930.118,A -85,B 0,C 180,E1 25640.957,E2 25640.957} C_VEL
LIN {X 0,Y 528.17,Z 922.742,A -85,B 0,C 180,E1 25638.867,E2 25638.867} C_VEL
LIN {X 0,Y 528.426,Z 913.471,A -85,B 0,C 180,E1 25636.765,E2 25636.765} C_VEL
LIN {X 0,Y 528.784,Z 902.721,A -85,B 0,C 180,E1 25634.762,E2 25634.762} C_VEL
LIN {X 0,Y 529.257,Z 890.574,A -85,B 0,C 180,E1 25632.86,E2 25632.86} C_VEL
LIN {X 0,Y 529.9,Z 876.258,A -85,B 0,C 180,E1 25630.967,E2 25630.967} C_VEL
LIN {X 0,Y 530.673,Z 860.322,A -85,B 0,C 180,E1 25629.191,E2 25629.191} C_VEL
LIN {X 0,Y 531.518,Z 843.6,A -85,B 0,C 180,E1 25627.62,E2 25627.62} C_VEL
LIN {X 0,Y 532.406,Z 826.191,A -85,B 0,C 180,E1 25626.245,E2 25626.245} C_VEL
LIN {X 0,Y 533.264,Z 808.05,A -85,B 0,C 180,E1 25625.047,E2 25625.047} C_VEL
LIN {X 0,Y 534.094,Z 788.925,A -85,B 0,C 180,E1 25624.019,E2 25624.019} C_VEL
LIN {X 0,Y 534.822,Z 769.45,A -85,B 0,C 180,E1 25623.191,E2 25623.191} C_VEL
LIN {X 0,Y 535.431,Z 749.152,A -85,B 0,C 180,E1 25622.536,E2 25622.536} C_VEL
LIN {X 0,Y 535.891,Z 727.87,A -85,B 0,C 180,E1 25622.065,E2 25622.065} C_VEL
LIN {X 0,Y 537.903,Z 538.471,A -85,B 0,C 180,E1 25619.25,E2 25619.25} C_VEL
LIN {X 0,Y 538.39,Z 481.884,A -85,B 0,C 180,E1 25618.375,E2 25618.375} C_VEL
LIN {X 0,Y 536.455,Z 469.655,A -85,B 0,C 180,E1 25618,E2 25618} C_VEL
LIN {X 0,Y 538.958,Z 419.99,A -85,B 0,C 180,E1 25614.313,E2 25614.313} C_VEL
LIN {X 0,Y 539.534,Z 405.968,A -85,B 0,C 180,E1 25613.231,E2 25613.231} C_VEL
LIN {X 0,Y 531.986,Z 389.177,A -85,B 0,C 180,E1 25611.088,E2 25611.088} C_VEL
LIN {X 0,Y 528.602,Z 381.668,A -85,B 0,C 180,E1 25610.067,E2 25610.067} C_VEL
LIN {X 0,Y 528.513,Z 381.2,A -85,B 0,C 180,E1 25609.825,E2 25609.825} C_VEL
LIN {X 0,Y 528.474,Z 381.21,A -85,B 0,C 180,E1 25606.596,E2 25606.596} C_VEL
LIN {X 0,Y 528.473,Z 381.218,A -85,B 0,C 180,E1 25603.079,E2 25603.079} C_VEL
LIN {X 0,Y 528.524,Z 381.2,A -85,B 0,C 180,E1 25599.749,E2 25599.749} C_VEL
LIN {X 0,Y 528.461,Z 381.198,A -85,B 0,C 180,E1 25596.448,E2 25596.448} C_VEL
LIN {X 0,Y 528.509,Z 381.217,A -85,B 0,C 180,E1 25593.06,E2 25593.06} C_VEL
LIN {X 0,Y 528.467,Z 381.19,A -85,B 0,C 180,E1 25589.841,E2 25589.841} C_VEL
LIN {X 0,Y 528.471,Z 381.214,A -85,B 0,C 180,E1 25586.399,E2 25586.399} C_VEL
LIN {X 0,Y 528.508,Z 381.215,A -85,B 0,C 180,E1 25583.155,E2 25583.155} C_VEL
LIN {X 0,Y 528.459,Z 381.216,A -85,B 0,C 180,E1 25579.89,E2 25579.89} C_VEL
LIN {X 0,Y 528.526,Z 381.215,A -85,B 0,C 180,E1 25576.599,E2 25576.599} C_VEL
LIN {X 0,Y 528.458,Z 381.216,A -85,B 0,C 180,E1 25573.346,E2 25573.346} C_VEL
LIN {X 0,Y 528.497,Z 381.217,A -85,B 0,C 180,E1 25570.024,E2 25570.024} C_VEL
LIN {X 0,Y 528.463,Z 381.21,A -85,B 0,C 180,E1 25566.846,E2 25566.846} C_VEL
LIN {X 0,Y 528.463,Z 381.214,A -85,B 0,C 180,E1 25563.363,E2 25563.363} C_VEL
LIN {X 0,Y 528.509,Z 381.212,A -85,B 0,C 180,E1 25560.109,E2 25560.109} C_VEL
LIN {X 0,Y 528.452,Z 381.214,A -85,B 0,C 180,E1 25556.855,E2 25556.855} C_VEL
LIN {X 0,Y 528.528,Z 381.214,A -85,B 0,C 180,E1 25553.592,E2 25553.592} C_VEL
LIN {X 0,Y 528.452,Z 381.217,A -85,B 0,C 180,E1 25550.306,E2 25550.306} C_VEL
LIN {X 0,Y 528.473,Z 381.191,A -85,B 0,C 180,E1 25546.878,E2 25546.878} C_VEL
LIN {X 0,Y 528.46,Z 381.216,A -85,B 0,C 180,E1 25543.852,E2 25543.852} C_VEL
LIN {X 0,Y 528.452,Z 381.194,A -85,B 0,C 180,E1 25540.319,E2 25540.319} C_VEL
LIN {X 0,Y 528.502,Z 381.217,A -85,B 0,C 180,E1 25537.124,E2 25537.124} C_VEL
LIN {X 0,Y 528.446,Z 381.203,A -85,B 0,C 180,E1 25533.842,E2 25533.842} C_VEL
LIN {X 0,Y 528.515,Z 381.201,A -85,B 0,C 180,E1 25530.537,E2 25530.537} C_VEL
LIN {X 0,Y 528.447,Z 381.22,A -85,B 0,C 180,E1 25527.35,E2 25527.35} C_VEL
LIN {X 0,Y 528.474,Z 381.201,A -85,B 0,C 180,E1 25523.957,E2 25523.957} C_VEL
LIN {X 0,Y 528.451,Z 381.197,A -85,B 0,C 180,E1 25520.873,E2 25520.873} C_VEL
LIN {X 0,Y 528.476,Z 381.451,A -85,B 0,C 180,E1 25519.06,E2 25519.06} C_VEL
LIN {X 0,Y 528.829,Z 382.851,A -85,B 0,C 180,E1 25518.856,E2 25518.856} C_VEL
LIN {X 0,Y 531.234,Z 387.075,A -85,B 0,C 180,E1 25518.35,E2 25518.35} C_VEL
LIN {X 0,Y 545.301,Z 413.275,A -85,B 0,C 180,E1 25515.473,E2 25515.473} C_VEL
LIN {X 0,Y 544.18,Z 466.354,A -85,B 0,C 180,E1 25512.698,E2 25512.698} C_VEL
LIN {X 0,Y 546.033,Z 481.407,A -85,B 0,C 180,E1 25512.256,E2 25512.256} C_VEL
LIN {X 0,Y 543.449,Z 684.962,A -85,B 0,C 180,E1 25509.024,E2 25509.024} C_VEL
LIN {X 0,Y 541.802,Z 816.31,A -85,B 0,C 180,E1 25506.963,E2 25506.963} C_VEL
LIN {X 0,Y 541.065,Z 839.477,A -85,B 0,C 180,E1 25506.413,E2 25506.413} C_VEL
LIN {X 0,Y 540.186,Z 861.095,A -85,B 0,C 180,E1 25505.719,E2 25505.719} C_VEL
LIN {X 0,Y 539.159,Z 882.386,A -85,B 0,C 180,E1 25504.833,E2 25504.833} C_VEL
LIN {X 0,Y 538.07,Z 902.212,A -85,B 0,C 180,E1 25503.837,E2 25503.837} C_VEL
LIN {X 0,Y 536.755,Z 923.239,A -85,B 0,C 180,E1 25502.571,E2 25502.571} C_VEL
LIN {X 0,Y 535.49,Z 943.405,A -85,B 0,C 180,E1 25501.146,E2 25501.146} C_VEL
LIN {X 0,Y 534.111,Z 963.271,A -85,B 0,C 180,E1 25499.495,E2 25499.495} C_VEL
LIN {X 0,Y 532.815,Z 982.788,A -85,B 0,C 180,E1 25497.614,E2 25497.614} C_VEL
LIN {X 0,Y 531.723,Z 999.659,A -85,B 0,C 180,E1 25495.746,E2 25495.746} C_VEL
LIN {X 0,Y 530.695,Z 1015.992,A -85,B 0,C 180,E1 25493.66,E2 25493.66} C_VEL
LIN {X 0,Y 529.868,Z 1030.925,A -85,B 0,C 180,E1 25491.474,E2 25491.474} C_VEL
LIN {X 0,Y 529.229,Z 1043.728,A -85,B 0,C 180,E1 25489.307,E2 25489.307} C_VEL
LIN {X 0,Y 528.699,Z 1056.05,A -85,B 0,C 180,E1 25486.879,E2 25486.879} C_VEL
LIN {X 0,Y 528.367,Z 1065.99,A -85,B 0,C 180,E1 25484.577,E2 25484.577} C_VEL
LIN {X 0,Y 528.124,Z 1074.7,A -85,B 0,C 180,E1 25482.131,E2 25482.131} C_VEL
LIN {X 0,Y 527.98,Z 1081.774,A -85,B 0,C 180,E1 25479.703,E2 25479.703} C_VEL
LIN {X 0,Y 527.92,Z 1086.841,A -85,B 0,C 180,E1 25477.4,E2 25477.4} C_VEL
LIN {X 0,Y 527.914,Z 1090.436,A -85,B 0,C 180,E1 25475.216,E2 25475.216} C_VEL
LIN {X 0,Y 527.909,Z 1093.056,A -85,B 0,C 180,E1 25472.605,E2 25472.605} C_VEL
LIN {X 0,Y 527.891,Z 1093.939,A -85,B 0,C 180,E1 25470.326,E2 25470.326} C_VEL
LIN {X 0,Y 527.914,Z 1093.324,A -85,B 0,C 180,E1 25467.829,E2 25467.829} C_VEL
LIN {X 0,Y 527.908,Z 1091.389,A -85,B 0,C 180,E1 25465.546,E2 25465.546} C_VEL
LIN {X 0,Y 527.91,Z 1087.667,A -85,B 0,C 180,E1 25463.038,E2 25463.038} C_VEL
LIN {X 0,Y 527.985,Z 1083.062,A -85,B 0,C 180,E1 25460.847,E2 25460.847} C_VEL
LIN {X 0,Y 528.101,Z 1076.117,A -85,B 0,C 180,E1 25458.312,E2 25458.312} C_VEL
LIN {X 0,Y 528.27,Z 1068.522,A -85,B 0,C 180,E1 25456.091,E2 25456.091} C_VEL
LIN {X 0,Y 528.601,Z 1058.396,A -85,B 0,C 180,E1 25453.63,E2 25453.63} C_VEL
LIN {X 0,Y 529.015,Z 1047.987,A -85,B 0,C 180,E1 25451.486,E2 25451.486} C_VEL
LIN {X 0,Y 529.663,Z 1034.46,A -85,B 0,C 180,E1 25449.097,E2 25449.097} C_VEL
LIN {X 0,Y 530.477,Z 1020.054,A -85,B 0,C 180,E1 25446.895,E2 25446.895} C_VEL
LIN {X 0,Y 531.406,Z 1004.33,A -85,B 0,C 180,E1 25444.825,E2 25444.825} C_VEL
LIN {X 0,Y 532.58,Z 986.116,A -85,B 0,C 180,E1 25442.736,E2 25442.736} C_VEL
LIN {X 0,Y 533.841,Z 967.898,A -85,B 0,C 180,E1 25440.92,E2 25440.92} C_VEL
LIN {X 0,Y 535.098,Z 948.56,A -85,B 0,C 180,E1 25439.263,E2 25439.263} C_VEL
LIN {X 0,Y 536.496,Z 927.724,A -85,B 0,C 180,E1 25437.727,E2 25437.727} C_VEL
LIN {X 0,Y 537.711,Z 907.809,A -85,B 0,C 180,E1 25436.477,E2 25436.477} C_VEL
LIN {X 0,Y 538.962,Z 886.239,A -85,B 0,C 180,E1 25435.347,E2 25435.347} C_VEL
LIN {X 0,Y 539.935,Z 866.97,A -85,B 0,C 180,E1 25434.511,E2 25434.511} C_VEL
LIN {X 0,Y 540.906,Z 843.306,A -85,B 0,C 180,E1 25433.695,E2 25433.695} C_VEL
LIN {X 0,Y 541.646,Z 821.905,A -85,B 0,C 180,E1 25433.151,E2 25433.151} C_VEL
LIN {X 0,Y 542.206,Z 789.732,A -85,B 0,C 180,E1 25432.601,E2 25432.601} C_VEL
LIN {X 0,Y 544.727,Z 581.594,A -85,B 0,C 180,E1 25429.347,E2 25429.347} C_VEL
LIN {X 0,Y 545.887,Z 478.81,A -85,B 0,C 180,E1 25427.685,E2 25427.685} C_VEL
LIN {X 0,Y 544.078,Z 464.717,A -85,B 0,C 180,E1 25427.236,E2 25427.236} C_VEL
LIN {X 0,Y 545.312,Z 412.859,A -85,B 0,C 180,E1 25424.505,E2 25424.505} C_VEL
LIN {X 0,Y 535.414,Z 394.816,A -85,B 0,C 180,E1 25422.533,E2 25422.533} C_VEL
LIN {X 0,Y 530.243,Z 385.322,A -85,B 0,C 180,E1 25421.442,E2 25421.442} C_VEL
LIN {X 0,Y 528.548,Z 381.845,A -85,B 0,C 180,E1 25421.027,E2 25421.027} C_VEL
LIN {X 0,Y 528.443,Z 381.221,A -85,B 0,C 180,E1 25420.75,E2 25420.75} C_VEL
LIN {X 0,Y 528.501,Z 381.217,A -85,B 0,C 180,E1 25417.53,E2 25417.53} C_VEL
LIN {X 0,Y 528.447,Z 381.209,A -85,B 0,C 180,E1 25414.321,E2 25414.321} C_VEL
LIN {X 0,Y 528.457,Z 381.196,A -85,B 0,C 180,E1 25410.846,E2 25410.846} C_VEL
LIN {X 0,Y 528.46,Z 381.22,A -85,B 0,C 180,E1 25407.861,E2 25407.861} C_VEL
LIN {X 0,Y 528.449,Z 381.211,A -85,B 0,C 180,E1 25404.36,E2 25404.36} C_VEL
LIN {X 0,Y 528.508,Z 381.203,A -85,B 0,C 180,E1 25401.142,E2 25401.142} C_VEL
LIN {X 0,Y 528.446,Z 381.211,A -85,B 0,C 180,E1 25397.849,E2 25397.849} C_VEL
LIN {X 0,Y 528.509,Z 381.198,A -85,B 0,C 180,E1 25394.573,E2 25394.573} C_VEL
LIN {X 0,Y 528.451,Z 381.205,A -85,B 0,C 180,E1 25391.348,E2 25391.348} C_VEL
LIN {X 0,Y 528.47,Z 381.209,A -85,B 0,C 180,E1 25387.938,E2 25387.938} C_VEL
LIN {X 0,Y 528.462,Z 381.216,A -85,B 0,C 180,E1 25384.884,E2 25384.884} C_VEL
LIN {X 0,Y 528.455,Z 381.214,A -85,B 0,C 180,E1 25381.409,E2 25381.409} C_VEL
LIN {X 0,Y 528.496,Z 381.218,A -85,B 0,C 180,E1 25378.265,E2 25378.265} C_VEL
LIN {X 0,Y 528.452,Z 381.217,A -85,B 0,C 180,E1 25375.007,E2 25375.007} C_VEL
LIN {X 0,Y 528.524,Z 381.211,A -85,B 0,C 180,E1 25371.733,E2 25371.733} C_VEL
LIN {X 0,Y 528.452,Z 381.211,A -85,B 0,C 180,E1 25368.43,E2 25368.43} C_VEL
LIN {X 0,Y 528.489,Z 381.211,A -85,B 0,C 180,E1 25365.09,E2 25365.09} C_VEL
LIN {X 0,Y 528.465,Z 381.216,A -85,B 0,C 180,E1 25361.923,E2 25361.923} C_VEL
LIN {X 0,Y 528.462,Z 381.211,A -85,B 0,C 180,E1 25358.466,E2 25358.466} C_VEL
LIN {X 0,Y 528.496,Z 381.216,A -85,B 0,C 180,E1 25355.284,E2 25355.284} C_VEL
LIN {X 0,Y 528.457,Z 381.215,A -85,B 0,C 180,E1 25352.016,E2 25352.016} C_VEL
LIN {X 0,Y 528.522,Z 381.192,A -85,B 0,C 180,E1 25348.771,E2 25348.771} C_VEL
LIN {X 0,Y 528.457,Z 381.214,A -85,B 0,C 180,E1 25345.528,E2 25345.528} C_VEL
LIN {X 0,Y 528.505,Z 381.213,A -85,B 0,C 180,E1 25342.196,E2 25342.196} C_VEL
LIN {X 0,Y 528.469,Z 381.218,A -85,B 0,C 180,E1 25341.792,E2 25341.792} C_VEL
LIN {X 0,Y 527.469,Z 381.346,A -85,B 0,C 180,E1 25340.958,E2 25340.958} C_VEL
LIN {X 0,Y 521.035,Z 382.122,A -85,B 0,C 180,E1 25338.55,E2 25338.55} C_VEL
LIN {X 0,Y 520.564,Z 382.187,A -85,B 0,C 180,E1 25338,E2 25338} C_VEL
LIN {X 0,Y 520.522,Z 382.186,A -85,B 0,C 180,E1 25334.827,E2 25334.827} C_VEL
LIN {X 0,Y 520.528,Z 382.186,A -85,B 0,C 180,E1 25331.318,E2 25331.318} C_VEL
LIN {X 0,Y 520.576,Z 382.542,A -85,B 0,C 180,E1 25330.653,E2 25330.653} C_VEL
LIN {X 0,Y 522.021,Z 385.88,A -85,B 0,C 180,E1 25330.161,E2 25330.161} C_VEL
LIN {X 0,Y 529.774,Z 402.487,A -85,B 0,C 180,E1 25327.916,E2 25327.916} C_VEL
LIN {X 0,Y 533.087,Z 410.466,A -85,B 0,C 180,E1 25326.924,E2 25326.924} C_VEL
LIN {X 0,Y 530.485,Z 456.272,A -85,B 0,C 180,E1 25323.457,E2 25323.457} C_VEL
LIN {X 0,Y 529.871,Z 470.551,A -85,B 0,C 180,E1 25322.423,E2 25322.423} C_VEL
LIN {X 0,Y 532.199,Z 485.596,A -85,B 0,C 180,E1 25321.986,E2 25321.986} C_VEL
LIN {X 0,Y 529.409,Z 701.019,A -85,B 0,C 180,E1 25318.709,E2 25318.709} C_VEL
LIN {X 0,Y 528.849,Z 734.846,A -85,B 0,C 180,E1 25318.15,E2 25318.15} C_VEL
LIN {X 0,Y 528.179,Z 754.944,A -85,B 0,C 180,E1 25317.617,E2 25317.617} C_VEL
LIN {X 0,Y 527.409,Z 775.372,A -85,B 0,C 180,E1 25316.882,E2 25316.882} C_VEL
LIN {X 0,Y 526.595,Z 794.013,A -85,B 0,C 180,E1 25316.015,E2 25316.015} C_VEL
LIN {X 0,Y 525.631,Z 813.051,A -85,B 0,C 180,E1 25314.919,E2 25314.919} C_VEL
LIN {X 0,Y 524.68,Z 831.148,A -85,B 0,C 180,E1 25313.65,E2 25313.65} C_VEL
LIN {X 0,Y 523.728,Z 848.316,A -85,B 0,C 180,E1 25312.21,E2 25312.21} C_VEL
LIN {X 0,Y 522.827,Z 864.492,A -85,B 0,C 180,E1 25310.603,E2 25310.603} C_VEL
LIN {X 0,Y 521.983,Z 880.004,A -85,B 0,C 180,E1 25308.772,E2 25308.772} C_VEL
LIN {X 0,Y 521.302,Z 893.818,A -85,B 0,C 180,E1 25306.835,E2 25306.835} C_VEL
LIN {X 0,Y 520.787,Z 905.395,A -85,B 0,C 180,E1 25304.908,E2 25304.908} C_VEL
LIN {X 0,Y 520.418,Z 915.642,A -85,B 0,C 180,E1 25302.878,E2 25302.878} C_VEL
LIN {X 0,Y 520.168,Z 924.497,A -85,B 0,C 180,E1 25300.746,E2 25300.746} C_VEL
LIN {X 0,Y 520.027,Z 931.567,A -85,B 0,C 180,E1 25298.625,E2 25298.625} C_VEL
LIN {X 0,Y 519.948,Z 937.41,A -85,B 0,C 180,E1 25296.293,E2 25296.293} C_VEL
LIN {X 0,Y 519.92,Z 941.181,A -85,B 0,C 180,E1 25294.08,E2 25294.08} C_VEL
LIN {X 0,Y 519.912,Z 943.345,A -85,B 0,C 180,E1 25291.874,E2 25291.874} C_VEL
LIN {X 0,Y 519.903,Z 943.949,A -85,B 0,C 180,E1 25289.669,E2 25289.669} C_VEL
LIN {X 0,Y 519.906,Z 942.991,A -85,B 0,C 180,E1 25287.465,E2 25287.465} C_VEL
LIN {X 0,Y 519.923,Z 940.355,A -85,B 0,C 180,E1 25285.257,E2 25285.257} C_VEL
LIN {X 0,Y 519.955,Z 936.092,A -85,B 0,C 180,E1 25283.042,E2 25283.042} C_VEL
LIN {X 0,Y 520.036,Z 930.116,A -85,B 0,C 180,E1 25280.817,E2 25280.817} C_VEL
LIN {X 0,Y 520.209,Z 922.739,A -85,B 0,C 180,E1 25278.694,E2 25278.694} C_VEL
LIN {X 0,Y 520.499,Z 913.469,A -85,B 0,C 180,E1 25276.559,E2 25276.559} C_VEL
LIN {X 0,Y 520.918,Z 902.476,A -85,B 0,C 180,E1 25274.483,E2 25274.483} C_VEL
LIN {X 0,Y 521.443,Z 890.568,A -85,B 0,C 180,E1 25272.595,E2 25272.595} C_VEL
LIN {X 0,Y 522.136,Z 876.839,A -85,B 0,C 180,E1 25270.746,E2 25270.746} C_VEL
LIN {X 0,Y 522.94,Z 862.037,A -85,B 0,C 180,E1 25269.05,E2 25269.05} C_VEL
LIN {X 0,Y 523.857,Z 845.973,A -85,B 0,C 180,E1 25267.486,E2 25267.486} C_VEL
LIN {X 0,Y 524.872,Z 828.047,A -85,B 0,C 180,E1 25266.021,E2 25266.021} C_VEL
LIN {X 0,Y 525.847,Z 809.324,A -85,B 0,C 180,E1 25264.753,E2 25264.753} C_VEL
LIN {X 0,Y 526.776,Z 790.04,A -85,B 0,C 180,E1 25263.692,E2 25263.692} C_VEL
LIN {X 0,Y 527.582,Z 770.91,A -85,B 0,C 180,E1 25262.854,E2 25262.854} C_VEL
LIN {X 0,Y 528.418,Z 748.218,A -85,B 0,C 180,E1 25262.096,E2 25262.096} C_VEL
LIN {X 0,Y 528.997,Z 727.646,A -85,B 0,C 180,E1 25261.621,E2 25261.621} C_VEL
LIN {X 0,Y 531.54,Z 540.309,A -85,B 0,C 180,E1 25258.751,E2 25258.751} C_VEL
LIN {X 0,Y 532.023,Z 483.291,A -85,B 0,C 180,E1 25257.872,E2 25257.872} C_VEL
LIN {X 0,Y 529.794,Z 469.391,A -85,B 0,C 180,E1 25257.429,E2 25257.429} C_VEL
LIN {X 0,Y 532.537,Z 419.705,A -85,B 0,C 180,E1 25253.695,E2 25253.695} C_VEL
LIN {X 0,Y 533.03,Z 409.822,A -85,B 0,C 180,E1 25252.928,E2 25252.928} C_VEL
LIN {X 0,Y 525.8,Z 393.89,A -85,B 0,C 180,E1 25250.851,E2 25250.851} C_VEL
LIN {X 0,Y 522.276,Z 386.211,A -85,B 0,C 180,E1 25249.806,E2 25249.806} C_VEL
LIN {X 0,Y 520.612,Z 382.705,A -85,B 0,C 180,E1 25249.291,E2 25249.291} C_VEL
LIN {X 0,Y 520.525,Z 382.183,A -85,B 0,C 180,E1 25249.017,E2 25249.017} C_VEL
LIN {X 0,Y 520.573,Z 382.179,A -85,B 0,C 180,E1 25245.642,E2 25245.642} C_VEL
LIN {X 0,Y 520.535,Z 382.201,A -85,B 0,C 180,E1 25242.393,E2 25242.393} C_VEL
LIN {X 0,Y 520.535,Z 382.209,A -85,B 0,C 180,E1 25238.911,E2 25238.911} C_VEL
LIN {X 0,Y 520.576,Z 382.176,A -85,B 0,C 180,E1 25235.589,E2 25235.589} C_VEL
LIN {X 0,Y 520.523,Z 382.203,A -85,B 0,C 180,E1 25232.277,E2 25232.277} C_VEL
LIN {X 0,Y 520.573,Z 382.183,A -85,B 0,C 180,E1 25228.948,E2 25228.948} C_VEL
LIN {X 0,Y 520.529,Z 382.201,A -85,B 0,C 180,E1 25225.725,E2 25225.725} C_VEL
LIN {X 0,Y 520.53,Z 382.2,A -85,B 0,C 180,E1 25222.202,E2 25222.202} C_VEL
LIN {X 0,Y 520.57,Z 382.2,A -85,B 0,C 180,E1 25218.942,E2 25218.942} C_VEL
LIN {X 0,Y 520.518,Z 382.202,A -85,B 0,C 180,E1 25215.601,E2 25215.601} C_VEL
LIN {X 0,Y 520.579,Z 382.201,A -85,B 0,C 180,E1 25212.31,E2 25212.31} C_VEL
LIN {X 0,Y 520.522,Z 382.205,A -85,B 0,C 180,E1 25209.063,E2 25209.063} C_VEL
LIN {X 0,Y 520.536,Z 382.207,A -85,B 0,C 180,E1 25205.622,E2 25205.622} C_VEL
LIN {X 0,Y 520.544,Z 382.201,A -85,B 0,C 180,E1 25202.422,E2 25202.422} C_VEL
LIN {X 0,Y 520.516,Z 382.204,A -85,B 0,C 180,E1 25199.01,E2 25199.01} C_VEL
LIN {X 0,Y 520.579,Z 382.197,A -85,B 0,C 180,E1 25195.705,E2 25195.705} C_VEL
LIN {X 0,Y 520.514,Z 382.2,A -85,B 0,C 180,E1 25192.495,E2 25192.495} C_VEL
LIN {X 0,Y 520.553,Z 382.196,A -85,B 0,C 180,E1 25189.151,E2 25189.151} C_VEL
LIN {X 0,Y 520.519,Z 382.185,A -85,B 0,C 180,E1 25185.943,E2 25185.943} C_VEL
LIN {X 0,Y 520.517,Z 382.2,A -85,B 0,C 180,E1 25182.448,E2 25182.448} C_VEL
LIN {X 0,Y 520.566,Z 382.183,A -85,B 0,C 180,E1 25179.187,E2 25179.187} C_VEL
LIN {X 0,Y 520.509,Z 382.199,A -85,B 0,C 180,E1 25175.969,E2 25175.969} C_VEL
LIN {X 0,Y 520.577,Z 382.196,A -85,B 0,C 180,E1 25172.675,E2 25172.675} C_VEL
LIN {X 0,Y 520.506,Z 382.184,A -85,B 0,C 180,E1 25169.4,E2 25169.4} C_VEL
LIN {X 0,Y 520.533,Z 382.198,A -85,B 0,C 180,E1 25166.016,E2 25166.016} C_VEL
LIN {X 0,Y 520.522,Z 382.21,A -85,B 0,C 180,E1 25162.861,E2 25162.861} C_VEL
LIN {X 0,Y 520.573,Z 382.401,A -85,B 0,C 180,E1 25159.857,E2 25159.857} C_VEL
LIN {X 0,Y 520.915,Z 383.865,A -85,B 0,C 180,E1 25159.642,E2 25159.642} C_VEL
LIN {X 0,Y 523.462,Z 388.55,A -85,B 0,C 180,E1 25159.069,E2 25159.069} C_VEL
LIN {X 0,Y 528.109,Z 397.066,A -85,B 0,C 180,E1 25158.062,E2 25158.062} C_VEL
LIN {X 0,Y 538.885,Z 417.155,A -85,B 0,C 180,E1 25155.837,E2 25155.837} C_VEL
LIN {X 0,Y 537.639,Z 466.291,A -85,B 0,C 180,E1 25153.241,E2 25153.241} C_VEL
LIN {X 0,Y 539.922,Z 482.761,A -85,B 0,C 180,E1 25152.786,E2 25152.786} C_VEL
LIN {X 0,Y 537.38,Z 674.099,A -85,B 0,C 180,E1 25149.735,E2 25149.735} C_VEL
LIN {X 0,Y 535.404,Z 816.331,A -85,B 0,C 180,E1 25147.479,E2 25147.479} C_VEL
LIN {X 0,Y 534.608,Z 839.345,A -85,B 0,C 180,E1 25146.929,E2 25146.929} C_VEL
LIN {X 0,Y 533.658,Z 860.559,A -85,B 0,C 180,E1 25146.245,E2 25146.245} C_VEL
LIN {X 0,Y 532.489,Z 882.383,A -85,B 0,C 180,E1 25145.334,E2 25145.334} C_VEL
LIN {X 0,Y 531.275,Z 902.569,A -85,B 0,C 180,E1 25144.309,E2 25144.309} C_VEL
LIN {X 0,Y 529.773,Z 924.136,A -85,B 0,C 180,E1 25142.991,E2 25142.991} C_VEL
LIN {X 0,Y 528.374,Z 944.183,A -85,B 0,C 180,E1 25141.549,E2 25141.549} C_VEL
LIN {X 0,Y 526.898,Z 963.268,A -85,B 0,C 180,E1 25139.939,E2 25139.939} C_VEL
LIN {X 0,Y 525.422,Z 983.136,A -85,B 0,C 180,E1 25137.998,E2 25137.998} C_VEL
LIN {X 0,Y 524.213,Z 999.658,A -85,B 0,C 180,E1 25136.142,E2 25136.142} C_VEL
LIN {X 0,Y 523.07,Z 1015.991,A -85,B 0,C 180,E1 25134.026,E2 25134.026} C_VEL
LIN {X 0,Y 522.121,Z 1031.237,A -85,B 0,C 180,E1 25131.757,E2 25131.757} C_VEL
LIN {X 0,Y 521.412,Z 1043.726,A -85,B 0,C 180,E1 25129.608,E2 25129.608} C_VEL
LIN {X 0,Y 520.824,Z 1055.804,A -85,B 0,C 180,E1 25127.196,E2 25127.196} C_VEL
LIN {X 0,Y 520.449,Z 1065.56,A -85,B 0,C 180,E1 25124.911,E2 25124.911} C_VEL
LIN {X 0,Y 520.163,Z 1074.345,A -85,B 0,C 180,E1 25122.432,E2 25122.432} C_VEL
LIN {X 0,Y 520.01,Z 1081.06,A -85,B 0,C 180,E1 25120.118,E2 25120.118} C_VEL
LIN {X 0,Y 519.939,Z 1086.635,A -85,B 0,C 180,E1 25117.625,E2 25117.625} C_VEL
LIN {X 0,Y 519.91,Z 1090.277,A -85,B 0,C 180,E1 25115.407,E2 25115.407} C_VEL
LIN {X 0,Y 519.893,Z 1092.919,A -85,B 0,C 180,E1 25112.866,E2 25112.866} C_VEL
LIN {X 0,Y 519.884,Z 1093.872,A -85,B 0,C 180,E1 25110.661,E2 25110.661} C_VEL
LIN {X 0,Y 519.907,Z 1093.526,A -85,B 0,C 180,E1 25108.126,E2 25108.126} C_VEL
LIN {X 0,Y 519.912,Z 1091.616,A -85,B 0,C 180,E1 25105.699,E2 25105.699} C_VEL
LIN {X 0,Y 519.917,Z 1088.08,A -85,B 0,C 180,E1 25103.152,E2 25103.152} C_VEL
LIN {X 0,Y 519.99,Z 1083.573,A -85,B 0,C 180,E1 25100.928,E2 25100.928} C_VEL
LIN {X 0,Y 520.101,Z 1077.175,A -85,B 0,C 180,E1 25098.467,E2 25098.467} C_VEL
LIN {X 0,Y 520.297,Z 1069.341,A -85,B 0,C 180,E1 25096.101,E2 25096.101} C_VEL
LIN {X 0,Y 520.643,Z 1059.938,A -85,B 0,C 180,E1 25093.717,E2 25093.717} C_VEL
LIN {X 0,Y 521.119,Z 1049.057,A -85,B 0,C 180,E1 25091.409,E2 25091.409} C_VEL
LIN {X 0,Y 521.829,Z 1035.859,A -85,B 0,C 180,E1 25089.004,E2 25089.004} C_VEL
LIN {X 0,Y 522.648,Z 1022.563,A -85,B 0,C 180,E1 25086.91,E2 25086.91} C_VEL
LIN {X 0,Y 523.695,Z 1006.725,A -85,B 0,C 180,E1 25084.741,E2 25084.741} C_VEL
LIN {X 0,Y 524.935,Z 989.959,A -85,B 0,C 180,E1 25082.733,E2 25082.733} C_VEL
LIN {X 0,Y 526.238,Z 972.177,A -85,B 0,C 180,E1 25080.895,E2 25080.895} C_VEL
LIN {X 0,Y 527.724,Z 952.256,A -85,B 0,C 180,E1 25079.106,E2 25079.106} C_VEL
LIN {X 0,Y 529.161,Z 933.152,A -85,B 0,C 180,E1 25077.63,E2 25077.63} C_VEL
LIN {X 0,Y 530.626,Z 911.825,A -85,B 0,C 180,E1 25076.229,E2 25076.229} C_VEL
LIN {X 0,Y 532.064,Z 890.06,A -85,B 0,C 180,E1 25075.029,E2 25075.029} C_VEL
LIN {X 0,Y 533.226,Z 869.3,A -85,B 0,C 180,E1 25074.1,E2 25074.1} C_VEL
LIN {X 0,Y 534.282,Z 847.802,A -85,B 0,C 180,E1 25073.317,E2 25073.317} C_VEL
LIN {X 0,Y 535.095,Z 825.314,A -85,B 0,C 180,E1 25072.712,E2 25072.712} C_VEL
LIN {X 0,Y 535.734,Z 799.299,A -85,B 0,C 180,E1 25072.229,E2 25072.229} C_VEL
LIN {X 0,Y 538.578,Z 587.829,A -85,B 0,C 180,E1 25068.891,E2 25068.891} C_VEL
LIN {X 0,Y 539.831,Z 480.848,A -85,B 0,C 180,E1 25067.177,E2 25067.177} C_VEL
LIN {X 0,Y 537.541,Z 464.593,A -85,B 0,C 180,E1 25066.693,E2 25066.693} C_VEL
LIN {X 0,Y 538.798,Z 416.774,A -85,B 0,C 180,E1 25064.135,E2 25064.135} C_VEL
LIN {X 0,Y 524.884,Z 390.957,A -85,B 0,C 180,E1 25061.231,E2 25061.231} C_VEL
LIN {X 0,Y 522.092,Z 386.075,A -85,B 0,C 180,E1 25060.627,E2 25060.627} C_VEL
LIN {X 0,Y 520.593,Z 382.566,A -85,B 0,C 180,E1 25060.19,E2 25060.19} C_VEL
LIN {X 0,Y 520.576,Z 382.177,A -85,B 0,C 180,E1 25059.76,E2 25059.76} C_VEL
LIN {X 0,Y 520.504,Z 382.201,A -85,B 0,C 180,E1 25056.547,E2 25056.547} C_VEL
LIN {X 0,Y 520.537,Z 382.209,A -85,B 0,C 180,E1 25053.125,E2 25053.125} C_VEL
LIN {X 0,Y 520.518,Z 382.188,A -85,B 0,C 180,E1 25049.962,E2 25049.962} C_VEL
LIN {X 0,Y 520.511,Z 382.194,A -85,B 0,C 180,E1 25046.465,E2 25046.465} C_VEL
LIN {X 0,Y 520.574,Z 382.201,A -85,B 0,C 180,E1 25043.187,E2 25043.187} C_VEL
LIN {X 0,Y 520.506,Z 382.182,A -85,B 0,C 180,E1 25039.877,E2 25039.877} C_VEL
LIN {X 0,Y 520.553,Z 382.205,A -85,B 0,C 180,E1 25036.515,E2 25036.515} C_VEL
LIN {X 0,Y 520.509,Z 382.181,A -85,B 0,C 180,E1 25033.44,E2 25033.44} C_VEL
LIN {X 0,Y 520.527,Z 382.204,A -85,B 0,C 180,E1 25029.955,E2 25029.955} C_VEL
LIN {X 0,Y 520.543,Z 382.199,A -85,B 0,C 180,E1 25026.753,E2 25026.753} C_VEL
LIN {X 0,Y 520.513,Z 382.202,A -85,B 0,C 180,E1 25023.414,E2 25023.414} C_VEL
LIN {X 0,Y 520.585,Z 382.196,A -85,B 0,C 180,E1 25020.11,E2 25020.11} C_VEL
LIN {X 0,Y 520.512,Z 382.203,A -85,B 0,C 180,E1 25016.806,E2 25016.806} C_VEL
LIN {X 0,Y 520.541,Z 382.199,A -85,B 0,C 180,E1 25013.382,E2 25013.382} C_VEL
LIN {X 0,Y 520.526,Z 382.207,A -85,B 0,C 180,E1 25010.268,E2 25010.268} C_VEL
LIN {X 0,Y 520.519,Z 382.206,A -85,B 0,C 180,E1 25006.786,E2 25006.786} C_VEL
LIN {X 0,Y 520.564,Z 382.204,A -85,B 0,C 180,E1 25003.599,E2 25003.599} C_VEL
LIN {X 0,Y 520.515,Z 382.205,A -85,B 0,C 180,E1 25000.24,E2 25000.24} C_VEL
LIN {X 0,Y 520.577,Z 382.204,A -85,B 0,C 180,E1 24996.928,E2 24996.928} C_VEL
LIN {X 0,Y 520.523,Z 382.203,A -85,B 0,C 180,E1 24993.658,E2 24993.658} C_VEL
LIN {X 0,Y 520.523,Z 382.178,A -85,B 0,C 180,E1 24990.165,E2 24990.165} C_VEL
LIN {X 0,Y 520.559,Z 382.206,A -85,B 0,C 180,E1 24986.942,E2 24986.942} C_VEL
LIN {X 0,Y 520.516,Z 382.184,A -85,B 0,C 180,E1 24983.59,E2 24983.59} C_VEL
LIN {X 0,Y 520.592,Z 382.19,A -85,B 0,C 180,E1 24980.37,E2 24980.37} C_VEL
LIN {X 0,Y 520.564,Z 382.187,A -85,B 0,C 180,E1 24978,E2 24978} C_VEL
LIN {X 0,Y 519.513,Z 382.333,A -85,B 0,C 180,E1 24977.152,E2 24977.152} C_VEL
LIN {X 0,Y 513.124,Z 383.107,A -85,B 0,C 180,E1 24974.771,E2 24974.771} C_VEL
LIN {X 0,Y 512.639,Z 383.165,A -85,B 0,C 180,E1 24974.15,E2 24974.15} C_VEL
LIN {X 0,Y 512.635,Z 383.404,A -85,B 0,C 180,E1 24971.499,E2 24971.499} C_VEL
LIN {X 0,Y 514.07,Z 386.917,A -85,B 0,C 180,E1 24970.955,E2 24970.955} C_VEL
LIN {X 0,Y 518.773,Z 396.737,A -85,B 0,C 180,E1 24969.561,E2 24969.561} C_VEL
LIN {X 0,Y 525.31,Z 410.975,A -85,B 0,C 180,E1 24967.645,E2 24967.645} C_VEL
LIN {X 0,Y 526.531,Z 413.839,A -85,B 0,C 180,E1 24967.282,E2 24967.282} C_VEL
LIN {X 0,Y 523.705,Z 460.03,A -85,B 0,C 180,E1 24963.751,E2 24963.751} C_VEL
LIN {X 0,Y 523.28,Z 470.621,A -85,B 0,C 180,E1 24962.99,E2 24962.99} C_VEL
LIN {X 0,Y 525.865,Z 486.724,A -85,B 0,C 180,E1 24962.505,E2 24962.505} C_VEL
LIN {X 0,Y 523.166,Z 694.351,A -85,B 0,C 180,E1 24959.347,E2 24959.347} C_VEL
LIN {X 0,Y 522.5,Z 735.072,A -85,B 0,C 180,E1 24958.683,E2 24958.683} C_VEL
LIN {X 0,Y 521.778,Z 755.214,A -85,B 0,C 180,E1 24958.149,E2 24958.149} C_VEL
LIN {X 0,Y 520.864,Z 773.533,A -85,B 0,C 180,E1 24957.467,E2 24957.467} C_VEL
LIN {X 0,Y 519.682,Z 792.873,A -85,B 0,C 180,E1 24956.536,E2 24956.536} C_VEL
LIN {X 0,Y 518.412,Z 811.408,A -85,B 0,C 180,E1 24955.413,E2 24955.413} C_VEL
LIN {X 0,Y 517.283,Z 830.421,A -85,B 0,C 180,E1 24954.07,E2 24954.07} C_VEL
LIN {X 0,Y 516.228,Z 847.536,A -85,B 0,C 180,E1 24952.628,E2 24952.628} C_VEL
LIN {X 0,Y 515.172,Z 864.499,A -85,B 0,C 180,E1 24950.923,E2 24950.923} C_VEL
LIN {X 0,Y 514.238,Z 880.009,A -85,B 0,C 180,E1 24949.066,E2 24949.066} C_VEL
LIN {X 0,Y 513.473,Z 893.821,A -85,B 0,C 180,E1 24947.1,E2 24947.1} C_VEL
LIN {X 0,Y 512.904,Z 905.398,A -85,B 0,C 180,E1 24945.143,E2 24945.143} C_VEL
LIN {X 0,Y 512.487,Z 915.645,A -85,B 0,C 180,E1 24943.08,E2 24943.08} C_VEL
LIN {X 0,Y 512.2,Z 924.5,A -85,B 0,C 180,E1 24940.915,E2 24940.915} C_VEL
LIN {X 0,Y 512.04,Z 931.569,A -85,B 0,C 180,E1 24938.761,E2 24938.761} C_VEL
LIN {X 0,Y 511.955,Z 937.159,A -85,B 0,C 180,E1 24936.504,E2 24936.504} C_VEL
LIN {X 0,Y 511.922,Z 941.024,A -85,B 0,C 180,E1 24934.256,E2 24934.256} C_VEL
LIN {X 0,Y 511.913,Z 943.345,A -85,B 0,C 180,E1 24931.903,E2 24931.903} C_VEL
LIN {X 0,Y 511.903,Z 943.949,A -85,B 0,C 180,E1 24929.664,E2 24929.664} C_VEL
LIN {X 0,Y 511.907,Z 942.99,A -85,B 0,C 180,E1 24927.425,E2 24927.425} C_VEL
LIN {X 0,Y 511.924,Z 940.353,A -85,B 0,C 180,E1 24925.182,E2 24925.182} C_VEL
LIN {X 0,Y 511.958,Z 936.091,A -85,B 0,C 180,E1 24922.932,E2 24922.932} C_VEL
LIN {X 0,Y 512.054,Z 930.114,A -85,B 0,C 180,E1 24920.673,E2 24920.673} C_VEL
LIN {X 0,Y 512.257,Z 922.575,A -85,B 0,C 180,E1 24918.476,E2 24918.476} C_VEL
LIN {X 0,Y 512.59,Z 913.085,A -85,B 0,C 180,E1 24916.265,E2 24916.265} C_VEL
LIN {X 0,Y 513.068,Z 902.075,A -85,B 0,C 180,E1 24914.167,E2 24914.167} C_VEL
LIN {X 0,Y 513.689,Z 889.79,A -85,B 0,C 180,E1 24912.206,E2 24912.206} C_VEL
LIN {X 0,Y 514.459,Z 876.087,A -85,B 0,C 180,E1 24910.353,E2 24910.353} C_VEL
LIN {X 0,Y 515.416,Z 860.359,A -85,B 0,C 180,E1 24908.551,E2 24908.551} C_VEL
LIN {X 0,Y 516.419,Z 844.111,A -85,B 0,C 180,E1 24906.977,E2 24906.977} C_VEL
LIN {X 0,Y 517.49,Z 826.977,A -85,B 0,C 180,E1 24905.576,E2 24905.576} C_VEL
LIN {X 0,Y 518.882,Z 804.62,A -85,B 0,C 180,E1 24904.061,E2 24904.061} C_VEL
LIN {X 0,Y 520.066,Z 787.323,A -85,B 0,C 180,E1 24903.079,E2 24903.079} C_VEL
LIN {X 0,Y 521.132,Z 768.696,A -85,B 0,C 180,E1 24902.241,E2 24902.241} C_VEL
LIN {X 0,Y 522.01,Z 749.356,A -85,B 0,C 180,E1 24901.588,E2 24901.588} C_VEL
LIN {X 0,Y 522.623,Z 728.855,A -85,B 0,C 180,E1 24901.108,E2 24901.108} C_VEL
LIN {X 0,Y 524.957,Z 560.256,A -85,B 0,C 180,E1 24898.514,E2 24898.514} C_VEL
LIN {X 0,Y 525.692,Z 484.666,A -85,B 0,C 180,E1 24897.357,E2 24897.357} C_VEL
LIN {X 0,Y 523.18,Z 469.472,A -85,B 0,C 180,E1 24896.867,E2 24896.867} C_VEL
LIN {X 0,Y 526.104,Z 420.446,A -85,B 0,C 180,E1 24893.141,E2 24893.141} C_VEL
LIN {X 0,Y 526.459,Z 413.605,A -85,B 0,C 180,E1 24892.602,E2 24892.602} C_VEL
LIN {X 0,Y 519.48,Z 398.304,A -85,B 0,C 180,E1 24890.568,E2 24890.568} C_VEL
LIN {X 0,Y 515.743,Z 390.435,A -85,B 0,C 180,E1 24889.461,E2 24889.461} C_VEL
LIN {X 0,Y 514.187,Z 387.064,A -85,B 0,C 180,E1 24888.981,E2 24888.981} C_VEL
LIN {X 0,Y 512.661,Z 383.511,A -85,B 0,C 180,E1 24888.439,E2 24888.439} C_VEL
LIN {X 0,Y 512.634,Z 383.186,A -85,B 0,C 180,E1 24887.708,E2 24887.708} C_VEL
LIN {X 0,Y 512.599,Z 383.179,A -85,B 0,C 180,E1 24884.446,E2 24884.446} C_VEL
LIN {X 0,Y 512.593,Z 383.17,A -85,B 0,C 180,E1 24880.95,E2 24880.95} C_VEL
LIN {X 0,Y 512.647,Z 383.183,A -85,B 0,C 180,E1 24877.624,E2 24877.624} C_VEL
LIN {X 0,Y 512.587,Z 383.191,A -85,B 0,C 180,E1 24874.201,E2 24874.201} C_VEL
LIN {X 0,Y 512.603,Z 383.164,A -85,B 0,C 180,E1 24870.734,E2 24870.734} C_VEL
LIN {X 0,Y 512.607,Z 383.191,A -85,B 0,C 180,E1 24867.534,E2 24867.534} C_VEL
LIN {X 0,Y 512.585,Z 383.195,A -85,B 0,C 180,E1 24864.091,E2 24864.091} C_VEL
LIN {X 0,Y 512.65,Z 383.189,A -85,B 0,C 180,E1 24860.792,E2 24860.792} C_VEL
LIN {X 0,Y 512.583,Z 383.193,A -85,B 0,C 180,E1 24857.472,E2 24857.472} C_VEL
LIN {X 0,Y 512.601,Z 383.196,A -85,B 0,C 180,E1 24853.997,E2 24853.997} C_VEL
LIN {X 0,Y 512.606,Z 383.185,A -85,B 0,C 180,E1 24850.793,E2 24850.793} C_VEL
LIN {X 0,Y 512.578,Z 383.188,A -85,B 0,C 180,E1 24847.397,E2 24847.397} C_VEL
LIN {X 0,Y 512.64,Z 383.187,A -85,B 0,C 180,E1 24844.139,E2 24844.139} C_VEL
LIN {X 0,Y 512.578,Z 383.193,A -85,B 0,C 180,E1 24840.783,E2 24840.783} C_VEL
LIN {X 0,Y 512.599,Z 383.193,A -85,B 0,C 180,E1 24837.317,E2 24837.317} C_VEL
LIN {X 0,Y 512.603,Z 383.194,A -85,B 0,C 180,E1 24834.067,E2 24834.067} C_VEL
LIN {X 0,Y 512.576,Z 383.196,A -85,B 0,C 180,E1 24830.683,E2 24830.683} C_VEL
LIN {X 0,Y 512.638,Z 383.159,A -85,B 0,C 180,E1 24827.383,E2 24827.383} C_VEL
LIN {X 0,Y 512.573,Z 383.194,A -85,B 0,C 180,E1 24824.089,E2 24824.089} C_VEL
LIN {X 0,Y 512.594,Z 383.164,A -85,B 0,C 180,E1 24820.635,E2 24820.635} C_VEL
LIN {X 0,Y 512.585,Z 383.195,A -85,B 0,C 180,E1 24817.523,E2 24817.523} C_VEL
LIN {X 0,Y 512.574,Z 383.172,A -85,B 0,C 180,E1 24814.061,E2 24814.061} C_VEL
LIN {X 0,Y 512.626,Z 383.183,A -85,B 0,C 180,E1 24810.816,E2 24810.816} C_VEL
LIN {X 0,Y 512.568,Z 383.199,A -85,B 0,C 180,E1 24807.559,E2 24807.559} C_VEL
LIN {X 0,Y 512.619,Z 383.168,A -85,B 0,C 180,E1 24804.187,E2 24804.187} C_VEL
LIN {X 0,Y 512.57,Z 383.171,A -85,B 0,C 180,E1 24800.93,E2 24800.93} C_VEL
LIN {X 0,Y 512.667,Z 383.655,A -85,B 0,C 180,E1 24800.623,E2 24800.623} C_VEL
LIN {X 0,Y 514.284,Z 387.119,A -85,B 0,C 180,E1 24800.171,E2 24800.171} C_VEL
LIN {X 0,Y 515.418,Z 389.199,A -85,B 0,C 180,E1 24799.906,E2 24799.906} C_VEL
LIN {X 0,Y 524.15,Z 405.259,A -85,B 0,C 180,E1 24797.967,E2 24797.967} C_VEL
LIN {X 0,Y 532.491,Z 420.91,A -85,B 0,C 180,E1 24796.217,E2 24796.217} C_VEL
LIN {X 0,Y 531.113,Z 466.311,A -85,B 0,C 180,E1 24793.784,E2 24793.784} C_VEL
LIN {X 0,Y 533.487,Z 484.248,A -85,B 0,C 180,E1 24793.277,E2 24793.277} C_VEL
LIN {X 0,Y 531.872,Z 630.711,A -85,B 0,C 180,E1 24790.986,E2 24790.986} C_VEL
LIN {X 0,Y 529.056,Z 816.082,A -85,B 0,C 180,E1 24788.013,E2 24788.013} C_VEL
LIN {X 0,Y 528.203,Z 839.081,A -85,B 0,C 180,E1 24787.462,E2 24787.462} C_VEL
LIN {X 0,Y 527.215,Z 859.483,A -85,B 0,C 180,E1 24786.803,E2 24786.803} C_VEL
LIN {X 0,Y 525.861,Z 882.38,A -85,B 0,C 180,E1 24785.847,E2 24785.847} C_VEL
LIN {X 0,Y 524.539,Z 902.572,A -85,B 0,C 180,E1 24784.813,E2 24784.813} C_VEL
LIN {X 0,Y 522.894,Z 924.132,A -85,B 0,C 180,E1 24783.481,E2 24783.481} C_VEL
LIN {X 0,Y 521.359,Z 943.97,A -85,B 0,C 180,E1 24782.042,E2 24782.042} C_VEL
LIN {X 0,Y 519.729,Z 963.266,A -85,B 0,C 180,E1 24780.395,E2 24780.395} C_VEL
LIN {X 0,Y 518.111,Z 982.785,A -85,B 0,C 180,E1 24778.468,E2 24778.468} C_VEL
LIN {X 0,Y 516.728,Z 999.657,A -85,B 0,C 180,E1 24776.55,E2 24776.55} C_VEL
LIN {X 0,Y 515.534,Z 1015.144,A -85,B 0,C 180,E1 24774.522,E2 24774.522} C_VEL
LIN {X 0,Y 514.478,Z 1030.219,A -85,B 0,C 180,E1 24772.27,E2 24772.27} C_VEL
LIN {X 0,Y 513.637,Z 1043.089,A -85,B 0,C 180,E1 24770.036,E2 24770.036} C_VEL
LIN {X 0,Y 512.95,Z 1055.805,A -85,B 0,C 180,E1 24767.469,E2 24767.469} C_VEL
LIN {X 0,Y 512.524,Z 1065.529,A -85,B 0,C 180,E1 24765.154,E2 24765.154} C_VEL
LIN {X 0,Y 512.196,Z 1074.538,A -85,B 0,C 180,E1 24762.567,E2 24762.567} C_VEL
LIN {X 0,Y 512.028,Z 1081.246,A -85,B 0,C 180,E1 24760.207,E2 24760.207} C_VEL
LIN {X 0,Y 511.954,Z 1086.635,A -85,B 0,C 180,E1 24757.745,E2 24757.745} C_VEL
LIN {X 0,Y 511.908,Z 1090.277,A -85,B 0,C 180,E1 24755.492,E2 24755.492} C_VEL
LIN {X 0,Y 511.891,Z 1092.919,A -85,B 0,C 180,E1 24752.911,E2 24752.911} C_VEL
LIN {X 0,Y 511.884,Z 1093.872,A -85,B 0,C 180,E1 24750.671,E2 24750.671} C_VEL
LIN {X 0,Y 511.908,Z 1093.526,A -85,B 0,C 180,E1 24748.097,E2 24748.097} C_VEL
LIN {X 0,Y 511.914,Z 1091.729,A -85,B 0,C 180,E1 24745.743,E2 24745.743} C_VEL
LIN {X 0,Y 511.925,Z 1088.494,A -85,B 0,C 180,E1 24743.27,E2 24743.27} C_VEL
LIN {X 0,Y 511.997,Z 1083.828,A -85,B 0,C 180,E1 24740.899,E2 24740.899} C_VEL
LIN {X 0,Y 512.123,Z 1077.516,A -85,B 0,C 180,E1 24738.399,E2 24738.399} C_VEL
LIN {X 0,Y 512.353,Z 1069.424,A -85,B 0,C 180,E1 24735.904,E2 24735.904} C_VEL
LIN {X 0,Y 512.746,Z 1059.937,A -85,B 0,C 180,E1 24733.459,E2 24733.459} C_VEL
LIN {X 0,Y 513.276,Z 1049.152,A -85,B 0,C 180,E1 24731.133,E2 24731.133} C_VEL
LIN {X 0,Y 514.074,Z 1035.857,A -85,B 0,C 180,E1 24728.672,E2 24728.672} C_VEL
LIN {X 0,Y 514.993,Z 1022.564,A -85,B 0,C 180,E1 24726.546,E2 24726.546} C_VEL
LIN {X 0,Y 516.171,Z 1006.724,A -85,B 0,C 180,E1 24724.346,E2 24724.346} C_VEL
LIN {X 0,Y 517.531,Z 989.987,A -85,B 0,C 180,E1 24722.313,E2 24722.313} C_VEL
LIN {X 0,Y 518.991,Z 972.175,A -85,B 0,C 180,E1 24720.449,E2 24720.449} C_VEL
LIN {X 0,Y 520.633,Z 952.257,A -85,B 0,C 180,E1 24718.637,E2 24718.637} C_VEL
LIN {X 0,Y 522.24,Z 932.895,A -85,B 0,C 180,E1 24717.127,E2 24717.127} C_VEL
LIN {X 0,Y 523.821,Z 911.822,A -85,B 0,C 180,E1 24715.73,E2 24715.73} C_VEL
LIN {X 0,Y 525.41,Z 890.064,A -85,B 0,C 180,E1 24714.52,E2 24714.52} C_VEL
LIN {X 0,Y 526.678,Z 869.197,A -85,B 0,C 180,E1 24713.578,E2 24713.578} C_VEL
LIN {X 0,Y 527.83,Z 847.546,A -85,B 0,C 180,E1 24712.785,E2 24712.785} C_VEL
LIN {X 0,Y 528.726,Z 825.313,A -85,B 0,C 180,E1 24712.184,E2 24712.184} C_VEL
LIN {X 0,Y 529.413,Z 799.299,A -85,B 0,C 180,E1 24711.697,E2 24711.697} C_VEL
LIN {X 0,Y 532.474,Z 589.206,A -85,B 0,C 180,E1 24708.353,E2 24708.353} C_VEL
LIN {X 0,Y 533.318,Z 481.723,A -85,B 0,C 180,E1 24706.67,E2 24706.67} C_VEL
LIN {X 0,Y 531.033,Z 464.446,A -85,B 0,C 180,E1 24706.14,E2 24706.14} C_VEL
LIN {X 0,Y 532.477,Z 420.898,A -85,B 0,C 180,E1 24703.784,E2 24703.784} C_VEL
LIN {X 0,Y 519.036,Z 395.87,A -85,B 0,C 180,E1 24700.917,E2 24700.917} C_VEL
LIN {X 0,Y 514.291,Z 387.13,A -85,B 0,C 180,E1 24699.83,E2 24699.83} C_VEL
LIN {X 0,Y 512.663,Z 383.637,A -85,B 0,C 180,E1 24699.377,E2 24699.377} C_VEL
LIN {X 0,Y 512.568,Z 383.171,A -85,B 0,C 180,E1 24699.055,E2 24699.055} C_VEL
LIN {X 0,Y 512.618,Z 383.169,A -85,B 0,C 180,E1 24695.813,E2 24695.813} C_VEL
LIN {X 0,Y 512.567,Z 383.199,A -85,B 0,C 180,E1 24692.441,E2 24692.441} C_VEL
LIN {X 0,Y 512.609,Z 383.188,A -85,B 0,C 180,E1 24689.057,E2 24689.057} C_VEL
LIN {X 0,Y 512.573,Z 383.172,A -85,B 0,C 180,E1 24685.909,E2 24685.909} C_VEL
LIN {X 0,Y 512.578,Z 383.196,A -85,B 0,C 180,E1 24682.357,E2 24682.357} C_VEL
LIN {X 0,Y 512.617,Z 383.163,A -85,B 0,C 180,E1 24679.128,E2 24679.128} C_VEL
LIN {X 0,Y 512.57,Z 383.195,A -85,B 0,C 180,E1 24675.848,E2 24675.848} C_VEL
LIN {X 0,Y 512.636,Z 383.158,A -85,B 0,C 180,E1 24672.617,E2 24672.617} C_VEL
LIN {X 0,Y 512.576,Z 383.194,A -85,B 0,C 180,E1 24669.234,E2 24669.234} C_VEL
LIN {X 0,Y 512.583,Z 383.193,A -85,B 0,C 180,E1 24665.709,E2 24665.709} C_VEL
LIN {X 0,Y 512.615,Z 383.193,A -85,B 0,C 180,E1 24662.459,E2 24662.459} C_VEL
LIN {X 0,Y 512.573,Z 383.194,A -85,B 0,C 180,E1 24659.105,E2 24659.105} C_VEL
LIN {X 0,Y 512.631,Z 383.189,A -85,B 0,C 180,E1 24655.749,E2 24655.749} C_VEL
LIN {X 0,Y 512.578,Z 383.188,A -85,B 0,C 180,E1 24652.49,E2 24652.49} C_VEL
LIN {X 0,Y 512.586,Z 383.187,A -85,B 0,C 180,E1 24648.979,E2 24648.979} C_VEL
LIN {X 0,Y 512.614,Z 383.192,A -85,B 0,C 180,E1 24645.773,E2 24645.773} C_VEL
LIN {X 0,Y 512.576,Z 383.194,A -85,B 0,C 180,E1 24642.401,E2 24642.401} C_VEL
LIN {X 0,Y 512.644,Z 383.188,A -85,B 0,C 180,E1 24639.088,E2 24639.088} C_VEL
LIN {X 0,Y 512.579,Z 383.196,A -85,B 0,C 180,E1 24635.818,E2 24635.818} C_VEL
LIN {X 0,Y 512.595,Z 383.192,A -85,B 0,C 180,E1 24632.322,E2 24632.322} C_VEL
LIN {X 0,Y 512.608,Z 383.164,A -85,B 0,C 180,E1 24629.12,E2 24629.12} C_VEL
LIN {X 0,Y 512.579,Z 383.192,A -85,B 0,C 180,E1 24625.685,E2 24625.685} C_VEL
LIN {X 0,Y 512.644,Z 383.181,A -85,B 0,C 180,E1 24622.36,E2 24622.36} C_VEL
LIN {X 0,Y 512.579,Z 383.172,A -85,B 0,C 180,E1 24619.188,E2 24619.188} C_VEL
LIN {X 0,Y 512.605,Z 383.183,A -85,B 0,C 180,E1 24615.709,E2 24615.709} C_VEL
LIN {X 0,Y 512.639,Z 383.165,A -85,B 0,C 180,E1 24614.15,E2 24614.15} C_VEL
LIN {X 0,Y 511.748,Z 383.304,A -85,B 0,C 180,E1 24613.545,E2 24613.545} C_VEL
LIN {X 0,Y 508.539,Z 384.441,A -85,B 0,C 180,E1 24612.648,E2 24612.648} C_VEL
LIN {X 0,Y 506.775,Z 386.485,A -85,B 0,C 180,E1 24612.034,E2 24612.034} C_VEL
LIN {X 0,Y 506.781,Z 388.94,A -85,B 0,C 180,E1 24611.616,E2 24611.616} C_VEL
LIN {X 0,Y 514.546,Z 405.37,A -85,B 0,C 180,E1 24609.253,E2 24609.253} C_VEL
LIN {X 0,Y 519.954,Z 417.812,A -85,B 0,C 180,E1 24607.602,E2 24607.602} C_VEL
LIN {X 0,Y 516.949,Z 463.847,A -85,B 0,C 180,E1 24604.052,E2 24604.052} C_VEL
LIN {X 0,Y 516.722,Z 470.535,A -85,B 0,C 180,E1 24603.578,E2 24603.578} C_VEL
LIN {X 0,Y 519.576,Z 487.89,A -85,B 0,C 180,E1 24603.035,E2 24603.035} C_VEL
LIN {X 0,Y 516.871,Z 695.274,A -85,B 0,C 180,E1 24599.882,E2 24599.882} C_VEL
LIN {X 0,Y 516.195,Z 735.963,A -85,B 0,C 180,E1 24599.217,E2 24599.217} C_VEL
LIN {X 0,Y 515.439,Z 756.068,A -85,B 0,C 180,E1 24598.681,E2 24598.681} C_VEL
LIN {X 0,Y 514.467,Z 774.431,A -85,B 0,C 180,E1 24597.992,E2 24597.992} C_VEL
LIN {X 0,Y 513.174,Z 793.935,A -85,B 0,C 180,E1 24597.045,E2 24597.045} C_VEL
LIN {X 0,Y 511.822,Z 811.805,A -85,B 0,C 180,E1 24595.95,E2 24595.95} C_VEL
LIN {X 0,Y 510.293,Z 829.723,A -85,B 0,C 180,E1 24594.611,E2 24594.611} C_VEL
LIN {X 0,Y 508.827,Z 846.133,A -85,B 0,C 180,E1 24593.127,E2 24593.127} C_VEL
LIN {X 0,Y 507.536,Z 864.506,A -85,B 0,C 180,E1 24591.253,E2 24591.253} C_VEL
LIN {X 0,Y 506.508,Z 880.014,A -85,B 0,C 180,E1 24589.368,E2 24589.368} C_VEL
LIN {X 0,Y 505.698,Z 893.055,A -85,B 0,C 180,E1 24587.49,E2 24587.49} C_VEL
LIN {X 0,Y 505.061,Z 904.766,A -85,B 0,C 180,E1 24585.501,E2 24585.501} C_VEL
LIN {X 0,Y 504.561,Z 915.648,A -85,B 0,C 180,E1 24583.29,E2 24583.29} C_VEL
LIN {X 0,Y 504.228,Z 924.75,A -85,B 0,C 180,E1 24581.019,E2 24581.019} C_VEL
LIN {X 0,Y 504.048,Z 931.874,A -85,B 0,C 180,E1 24578.786,E2 24578.786} C_VEL
LIN {X 0,Y 503.958,Z 937.414,A -85,B 0,C 180,E1 24576.493,E2 24576.493} C_VEL
LIN {X 0,Y 503.922,Z 941.184,A -85,B 0,C 180,E1 24574.21,E2 24574.21} C_VEL
LIN {X 0,Y 503.913,Z 943.345,A -85,B 0,C 180,E1 24571.933,E2 24571.933} C_VEL
LIN {X 0,Y 503.903,Z 943.949,A -85,B 0,C 180,E1 24569.659,E2 24569.659} C_VEL
LIN {X 0,Y 503.907,Z 942.99,A -85,B 0,C 180,E1 24567.384,E2 24567.384} C_VEL
LIN {X 0,Y 503.924,Z 940.352,A -85,B 0,C 180,E1 24565.106,E2 24565.106} C_VEL
LIN {X 0,Y 503.962,Z 936.089,A -85,B 0,C 180,E1 24562.82,E2 24562.82} C_VEL
LIN {X 0,Y 504.075,Z 930.112,A -85,B 0,C 180,E1 24560.524,E2 24560.524} C_VEL
LIN {X 0,Y 504.298,Z 922.732,A -85,B 0,C 180,E1 24558.332,E2 24558.332} C_VEL
LIN {X 0,Y 504.655,Z 913.452,A -85,B 0,C 180,E1 24556.126,E2 24556.126} C_VEL
LIN {X 0,Y 505.171,Z 902.709,A -85,B 0,C 180,E1 24554.031,E2 24554.031} C_VEL
LIN {X 0,Y 505.851,Z 890.555,A -85,B 0,C 180,E1 24552.04,E2 24552.04} C_VEL
LIN {X 0,Y 506.693,Z 877.008,A -85,B 0,C 180,E1 24550.159,E2 24550.159} C_VEL
LIN {X 0,Y 507.699,Z 862.018,A -85,B 0,C 180,E1 24548.39,E2 24548.39} C_VEL
LIN {X 0,Y 509.192,Z 841.954,A -85,B 0,C 180,E1 24546.385,E2 24546.385} C_VEL
LIN {X 0,Y 510.695,Z 824.941,A -85,B 0,C 180,E1 24544.92,E2 24544.92} C_VEL
LIN {X 0,Y 512.209,Z 806.892,A -85,B 0,C 180,E1 24543.637,E2 24543.637} C_VEL
LIN {X 0,Y 513.554,Z 789.033,A -85,B 0,C 180,E1 24542.599,E2 24542.599} C_VEL
LIN {X 0,Y 514.718,Z 770.191,A -85,B 0,C 180,E1 24541.738,E2 24541.738} C_VEL
LIN {X 0,Y 515.656,Z 750.916,A -85,B 0,C 180,E1 24541.075,E2 24541.075} C_VEL
LIN {X 0,Y 516.307,Z 730.5,A -85,B 0,C 180,E1 24540.587,E2 24540.587} C_VEL
LIN {X 0,Y 518.528,Z 571.798,A -85,B 0,C 180,E1 24538.139,E2 24538.139} C_VEL
LIN {X 0,Y 519.414,Z 486.136,A -85,B 0,C 180,E1 24536.832,E2 24536.832} C_VEL
LIN {X 0,Y 516.616,Z 469.58,A -85,B 0,C 180,E1 24536.291,E2 24536.291} C_VEL
LIN {X 0,Y 519.678,Z 421.776,A -85,B 0,C 180,E1 24532.619,E2 24532.619} C_VEL
LIN {X 0,Y 519.793,Z 417.22,A -85,B 0,C 180,E1 24532.241,E2 24532.241} C_VEL
LIN {X 0,Y 512.35,Z 400.557,A -85,B 0,C 180,E1 24529.994,E2 24529.994} C_VEL
LIN {X 0,Y 506.113,Z 387.795,A -85,B 0,C 180,E1 24528.107,E2 24528.107} C_VEL
LIN {X 0,Y 504.726,Z 384.479,A -85,B 0,C 180,E1 24527.579,E2 24527.579} C_VEL
LIN {X 0,Y 504.705,Z 384.152,A -85,B 0,C 180,E1 24525.82,E2 24525.82} C_VEL
LIN {X 0,Y 504.652,Z 384.178,A -85,B 0,C 180,E1 24522.502,E2 24522.502} C_VEL
LIN {X 0,Y 504.659,Z 384.187,A -85,B 0,C 180,E1 24518.907,E2 24518.907} C_VEL
LIN {X 0,Y 504.701,Z 384.15,A -85,B 0,C 180,E1 24515.483,E2 24515.483} C_VEL
LIN {X 0,Y 504.646,Z 384.181,A -85,B 0,C 180,E1 24512.207,E2 24512.207} C_VEL
LIN {X 0,Y 504.677,Z 384.163,A -85,B 0,C 180,E1 24508.779,E2 24508.779} C_VEL
LIN {X 0,Y 504.669,Z 384.176,A -85,B 0,C 180,E1 24505.463,E2 24505.463} C_VEL
LIN {X 0,Y 504.645,Z 384.178,A -85,B 0,C 180,E1 24501.988,E2 24501.988} C_VEL
LIN {X 0,Y 504.703,Z 384.174,A -85,B 0,C 180,E1 24498.6,E2 24498.6} C_VEL
LIN {X 0,Y 504.648,Z 384.179,A -85,B 0,C 180,E1 24495.225,E2 24495.225} C_VEL
LIN {X 0,Y 504.645,Z 384.176,A -85,B 0,C 180,E1 24491.66,E2 24491.66} C_VEL
LIN {X 0,Y 504.706,Z 384.177,A -85,B 0,C 180,E1 24488.316,E2 24488.316} C_VEL
LIN {X 0,Y 504.639,Z 384.184,A -85,B 0,C 180,E1 24485.002,E2 24485.002} C_VEL
LIN {X 0,Y 504.67,Z 384.184,A -85,B 0,C 180,E1 24481.59,E2 24481.59} C_VEL
LIN {X 0,Y 504.653,Z 384.181,A -85,B 0,C 180,E1 24478.411,E2 24478.411} C_VEL
LIN {X 0,Y 504.639,Z 384.185,A -85,B 0,C 180,E1 24474.885,E2 24474.885} C_VEL
LIN {X 0,Y 504.705,Z 384.173,A -85,B 0,C 180,E1 24471.57,E2 24471.57} C_VEL
LIN {X 0,Y 504.636,Z 384.166,A -85,B 0,C 180,E1 24468.179,E2 24468.179} C_VEL
LIN {X 0,Y 504.644,Z 384.184,A -85,B 0,C 180,E1 24464.604,E2 24464.604} C_VEL
LIN {X 0,Y 504.685,Z 384.153,A -85,B 0,C 180,E1 24461.262,E2 24461.262} C_VEL
LIN {X 0,Y 504.632,Z 384.185,A -85,B 0,C 180,E1 24457.886,E2 24457.886} C_VEL
LIN {X 0,Y 504.672,Z 384.152,A -85,B 0,C 180,E1 24454.538,E2 24454.538} C_VEL
LIN {X 0,Y 504.64,Z 384.187,A -85,B 0,C 180,E1 24451.349,E2 24451.349} C_VEL
LIN {X 0,Y 504.635,Z 384.177,A -85,B 0,C 180,E1 24447.784,E2 24447.784} C_VEL
LIN {X 0,Y 504.683,Z 384.153,A -85,B 0,C 180,E1 24444.515,E2 24444.515} C_VEL
LIN {X 0,Y 504.659,Z 384.344,A -85,B 0,C 180,E1 24441.578,E2 24441.578} C_VEL
LIN {X 0,Y 505.004,Z 385.789,A -85,B 0,C 180,E1 24441.343,E2 24441.343} C_VEL
LIN {X 0,Y 507.465,Z 389.954,A -85,B 0,C 180,E1 24440.768,E2 24440.768} C_VEL
LIN {X 0,Y 516.913,Z 407.448,A -85,B 0,C 180,E1 24438.584,E2 24438.584} C_VEL
LIN {X 0,Y 526.11,Z 424.806,A -85,B 0,C 180,E1 24436.598,E2 24436.598} C_VEL
LIN {X 0,Y 524.65,Z 466.441,A -85,B 0,C 180,E1 24434.336,E2 24434.336} C_VEL
LIN {X 0,Y 527.108,Z 485.648,A -85,B 0,C 180,E1 24433.783,E2 24433.783} C_VEL
LIN {X 0,Y 525.058,Z 671.48,A -85,B 0,C 180,E1 24430.882,E2 24430.882} C_VEL
LIN {X 0,Y 522.761,Z 815.503,A -85,B 0,C 180,E1 24428.566,E2 24428.566} C_VEL
LIN {X 0,Y 521.85,Z 838.688,A -85,B 0,C 180,E1 24428.011,E2 24428.011} C_VEL
LIN {X 0,Y 520.82,Z 858.469,A -85,B 0,C 180,E1 24427.371,E2 24427.371} C_VEL
LIN {X 0,Y 519.337,Z 881.54,A -85,B 0,C 180,E1 24426.414,E2 24426.414} C_VEL
LIN {X 0,Y 517.842,Z 902.575,A -85,B 0,C 180,E1 24425.33,E2 24425.33} C_VEL
LIN {X 0,Y 516.141,Z 923.229,A -85,B 0,C 180,E1 24424.045,E2 24424.045} C_VEL
LIN {X 0,Y 514.407,Z 943.414,A -85,B 0,C 180,E1 24422.576,E2 24422.576} C_VEL
LIN {X 0,Y 512.673,Z 962.415,A -85,B 0,C 180,E1 24420.942,E2 24420.942} C_VEL
LIN {X 0,Y 510.957,Z 981.119,A -85,B 0,C 180,E1 24419.096,E2 24419.096} C_VEL
LIN {X 0,Y 509.469,Z 997.63,A -85,B 0,C 180,E1 24417.212,E2 24417.212} C_VEL
LIN {X 0,Y 508.036,Z 1014.297,A -85,B 0,C 180,E1 24415.033,E2 24415.033} C_VEL
LIN {X 0,Y 506.836,Z 1029.506,A -85,B 0,C 180,E1 24412.747,E2 24412.747} C_VEL
LIN {X 0,Y 505.851,Z 1043.087,A -85,B 0,C 180,E1 24410.358,E2 24410.358} C_VEL
LIN {X 0,Y 505.084,Z 1055.807,A -85,B 0,C 180,E1 24407.75,E2 24407.75} C_VEL
LIN {X 0,Y 504.602,Z 1065.528,A -85,B 0,C 180,E1 24405.398,E2 24405.398} C_VEL
LIN {X 0,Y 504.248,Z 1074.346,A -85,B 0,C 180,E1 24402.831,E2 24402.831} C_VEL
LIN {X 0,Y 504.069,Z 1080.866,A -85,B 0,C 180,E1 24400.515,E2 24400.515} C_VEL
LIN {X 0,Y 503.967,Z 1086.635,A -85,B 0,C 180,E1 24397.868,E2 24397.868} C_VEL
LIN {X 0,Y 503.907,Z 1090.278,A -85,B 0,C 180,E1 24395.58,E2 24395.58} C_VEL
LIN {X 0,Y 503.889,Z 1092.919,A -85,B 0,C 180,E1 24392.957,E2 24392.957} C_VEL
LIN {X 0,Y 503.884,Z 1093.872,A -85,B 0,C 180,E1 24390.682,E2 24390.682} C_VEL
LIN {X 0,Y 503.908,Z 1093.526,A -85,B 0,C 180,E1 24388.067,E2 24388.067} C_VEL
LIN {X 0,Y 503.912,Z 1091.729,A -85,B 0,C 180,E1 24385.676,E2 24385.676} C_VEL
LIN {X 0,Y 503.923,Z 1088.494,A -85,B 0,C 180,E1 24383.163,E2 24383.163} C_VEL
LIN {X 0,Y 504.003,Z 1083.828,A -85,B 0,C 180,E1 24380.753,E2 24380.753} C_VEL
LIN {X 0,Y 504.157,Z 1077.516,A -85,B 0,C 180,E1 24378.213,E2 24378.213} C_VEL
LIN {X 0,Y 504.423,Z 1069.343,A -85,B 0,C 180,E1 24375.654,E2 24375.654} C_VEL
LIN {X 0,Y 504.859,Z 1059.936,A -85,B 0,C 180,E1 24373.193,E2 24373.193} C_VEL
LIN {X 0,Y 505.456,Z 1049.153,A -85,B 0,C 180,E1 24370.83,E2 24370.83} C_VEL
LIN {X 0,Y 506.344,Z 1035.855,A -85,B 0,C 180,E1 24368.33,E2 24368.33} C_VEL
LIN {X 0,Y 507.391,Z 1022.186,A -85,B 0,C 180,E1 24366.113,E2 24366.113} C_VEL
LIN {X 0,Y 508.711,Z 1006.26,A -85,B 0,C 180,E1 24363.879,E2 24363.879} C_VEL
LIN {X 0,Y 510.212,Z 989.435,A -85,B 0,C 180,E1 24361.817,E2 24361.817} C_VEL
LIN {X 0,Y 511.775,Z 972.172,A -85,B 0,C 180,E1 24359.99,E2 24359.99} C_VEL
LIN {X 0,Y 513.587,Z 952.253,A -85,B 0,C 180,E1 24358.157,E2 24358.157} C_VEL
LIN {X 0,Y 515.259,Z 933.703,A -85,B 0,C 180,E1 24356.69,E2 24356.69} C_VEL
LIN {X 0,Y 516.986,Z 912.833,A -85,B 0,C 180,E1 24355.28,E2 24355.28} C_VEL
LIN {X 0,Y 518.608,Z 892.41,A -85,B 0,C 180,E1 24354.119,E2 24354.119} C_VEL
LIN {X 0,Y 520.087,Z 870.602,A -85,B 0,C 180,E1 24353.106,E2 24353.106} C_VEL
LIN {X 0,Y 521.291,Z 850.049,A -85,B 0,C 180,E1 24352.332,E2 24352.332} C_VEL
LIN {X 0,Y 522.317,Z 827.163,A -85,B 0,C 180,E1 24351.686,E2 24351.686} C_VEL
LIN {X 0,Y 523.072,Z 803.768,A -85,B 0,C 180,E1 24351.223,E2 24351.223} C_VEL
LIN {X 0,Y 525.168,Z 658.568,A -85,B 0,C 180,E1 24348.921,E2 24348.921} C_VEL
LIN {X 0,Y 527.092,Z 486.731,A -85,B 0,C 180,E1 24346.235,E2 24346.235} C_VEL
LIN {X 0,Y 526.756,Z 481.676,A -85,B 0,C 180,E1 24346.117,E2 24346.117} C_VEL
LIN {X 0,Y 524.558,Z 465.009,A -85,B 0,C 180,E1 24345.61,E2 24345.61} C_VEL
LIN {X 0,Y 526.093,Z 424.794,A -85,B 0,C 180,E1 24343.403,E2 24343.403} C_VEL
LIN {X 0,Y 513.705,Z 401.489,A -85,B 0,C 180,E1 24340.694,E2 24340.694} C_VEL
LIN {X 0,Y 508.771,Z 392.446,A -85,B 0,C 180,E1 24339.548,E2 24339.548} C_VEL
LIN {X 0,Y 506.559,Z 388.454,A -85,B 0,C 180,E1 24339.024,E2 24339.024} C_VEL
LIN {X 0,Y 504.783,Z 385.027,A -85,B 0,C 180,E1 24338.571,E2 24338.571} C_VEL
LIN {X 0,Y 504.644,Z 384.184,A -85,B 0,C 180,E1 24338.316,E2 24338.316} C_VEL
